C03602=1038.319,72.260,-89.888,169.485,39.498,157.426
C03603=1038.313,72.011,-89.869,169.482,39.498,157.426
C03604=1038.308,71.762,-89.852,169.480,39.497,157.426
C03605=1038.301,71.513,-89.833,169.478,39.498,157.426
C03606=1038.295,71.263,-89.815,169.476,39.497,157.425
C03607=1038.289,71.014,-89.797,169.474,39.497,157.425
C03608=1038.282,70.764,-89.779,169.472,39.497,157.425
C03609=1038.276,70.516,-89.761,169.471,39.496,157.425
C03610=1038.270,70.266,-89.743,169.469,39.496,157.425
C03611=1038.263,70.017,-89.724,169.467,39.496,157.425
C03612=1038.257,69.767,-89.706,169.465,39.495,157.425
C03613=1038.252,69.518,-89.689,169.462,39.495,157.425
C03614=1038.245,69.269,-89.670,169.460,39.495,157.425
C03615=1038.238,69.020,-89.653,169.458,39.495,157.424
C03616=1038.232,68.771,-89.634,169.456,39.494,157.424
C03617=1038.226,68.521,-89.616,169.454,39.494,157.424
C03618=1038.220,68.272,-89.599,169.452,39.494,157.424
C03619=1038.213,68.023,-89.581,169.450,39.494,157.424
C03620=1038.207,67.773,-89.563,169.448,39.493,157.424
C03621=1038.201,67.524,-89.545,169.446,39.493,157.424
C03622=1038.194,67.275,-89.527,169.444,39.493,157.424
C03623=1038.188,67.026,-89.509,169.441,39.493,157.423
C03624=1038.182,66.776,-89.491,169.439,39.493,157.423
C03625=1038.176,66.527,-89.473,169.438,39.492,157.423
C03626=1038.169,66.277,-89.455,169.436,39.492,157.423
C03627=1038.163,66.028,-89.438,169.434,39.492,157.423
C03628=1038.157,65.779,-89.419,169.432,39.491,157.423
C03629=1038.150,65.530,-89.402,169.430,39.492,157.423
C03630=1038.144,65.280,-89.384,169.428,39.491,157.423
C03631=1038.138,65.031,-89.366,169.426,39.491,157.423
C03632=1038.131,64.782,-89.348,169.424,39.491,157.423
C03633=1038.125,64.532,-89.330,169.421,39.490,157.422
C03634=1038.120,64.283,-89.313,169.419,39.490,157.422
C03635=1038.113,64.034,-89.295,169.417,39.490,157.422
C03636=1038.106,63.785,-89.277,169.415,39.489,157.422
C03637=1038.099,63.535,-89.259,169.413,39.490,157.422
C03638=1038.094,63.286,-89.242,169.411,39.489,157.422
C03639=1038.087,63.037,-89.224,169.409,39.489,157.422
C03640=1038.080,62.788,-89.207,169.407,39.489,157.422
C03641=1038.074,62.538,-89.189,169.405,39.489,157.422
C03642=1038.068,62.289,-89.172,169.403,39.488,157.421
C03643=1038.061,62.040,-89.154,169.401,39.489,157.421
C03644=1038.055,61.791,-89.136,169.399,39.488,157.421
C03645=1038.048,61.541,-89.119,169.397,39.488,157.421
C03646=1038.042,61.292,-89.101,169.394,39.488,157.421
C03647=1038.035,61.005,-89.081,169.392,39.488,157.421
C03648=1038.028,60.719,-89.061,169.390,39.487,157.421
C03649=1038.019,60.433,-89.041,169.387,39.488,157.421
C03650=1038.012,60.147,-89.021,169.385,39.487,157.421
C03651=1038.006,59.897,-89.003,169.383,39.487,157.421
C03652=1037.999,59.648,-88.986,169.381,39.487,157.420
C03653=1037.994,59.399,-88.969,169.379,39.487,157.420
C03654=1037.987,59.150,-88.951,169.377,39.487,157.420
C03655=1037.980,58.900,-88.934,169.375,39.487,157.420
C03656=1037.974,58.650,-88.916,169.373,39.486,157.420
C03657=1037.968,58.402,-88.899,169.370,39.486,157.420
C03658=1037.961,58.152,-88.882,169.368,39.486,157.420
C03659=1037.955,57.902,-88.864,169.366,39.486,157.420
C03660=1037.949,57.654,-88.847,169.364,39.486,157.420
C03661=1037.942,57.404,-88.829,169.362,39.486,157.419
C03662=1037.936,57.155,-88.812,169.360,39.485,157.419
C03663=1037.929,56.906,-88.794,169.358,39.485,157.419
C03664=1037.923,56.656,-88.777,169.357,39.485,157.419
C03665=1037.917,56.407,-88.760,169.355,39.485,157.419
C03666=1037.910,56.158,-88.742,169.353,39.485,157.419
C03667=1037.904,55.908,-88.724,169.351,39.485,157.419
C03668=1037.898,55.660,-88.707,169.349,39.484,157.419
C03669=1037.891,55.410,-88.690,169.347,39.484,157.419
C03670=1037.885,55.161,-88.672,169.344,39.484,157.419
C03671=1037.878,54.912,-88.655,169.342,39.483,157.418
C03672=1037.872,54.662,-88.638,169.340,39.484,157.418
C03673=1037.866,54.413,-88.620,169.338,39.483,157.418
C03674=1037.860,54.163,-88.604,169.336,39.483,157.418
C03675=1037.853,53.914,-88.587,169.334,39.483,157.418
C03676=1037.847,53.665,-88.569,169.332,39.483,157.418
C03677=1037.840,53.415,-88.551,169.330,39.482,157.418
C03678=1037.834,53.166,-88.534,169.328,39.483,157.418
C03679=1037.828,52.917,-88.516,169.326,39.482,157.418
C03680=1037.822,52.668,-88.499,169.324,39.482,157.418
C03681=1037.815,52.418,-88.483,169.321,39.482,157.417
C03682=1037.810,52.169,-88.465,169.319,39.481,157.417
C03683=1037.803,51.919,-88.448,169.317,39.481,157.417
C03684=1037.796,51.671,-88.431,169.315,39.481,157.417
C03685=1037.790,51.421,-88.413,169.313,39.481,157.417
C03686=1037.784,51.172,-88.396,169.311,39.481,157.417
C03687=1037.778,50.922,-88.379,169.309,39.481,157.417
C03688=1037.771,50.672,-88.361,169.307,39.480,157.417
C03689=1037.765,50.424,-88.345,169.305,39.480,157.417
C03690=1037.758,50.174,-88.327,169.303,39.480,157.416
C03691=1037.753,49.925,-88.310,169.300,39.479,157.416
C03692=1037.746,49.675,-88.293,169.298,39.480,157.416
C03693=1037.740,49.427,-88.276,169.296,39.479,157.416
C03694=1037.734,49.177,-88.258,169.294,39.479,157.416
C03695=1037.728,48.927,-88.242,169.293,39.479,157.416
C03696=1037.721,48.678,-88.224,169.291,39.478,157.416
C03697=1037.716,48.429,-88.207,169.289,39.478,157.416
C03698=1037.709,48.180,-88.190,169.287,39.478,157.415
C03699=1037.703,47.930,-88.173,169.285,39.478,157.415
C03700=1037.697,47.681,-88.156,169.283,39.478,157.415
C03701=1037.690,47.432,-88.138,169.280,39.477,157.415
C03702=1037.684,47.182,-88.122,169.278,39.477,157.415
C03703=1037.678,46.933,-88.104,169.276,39.477,157.415
C03704=1037.672,46.684,-88.087,169.274,39.477,157.415
C03705=1037.665,46.434,-88.071,169.272,39.476,157.415
C03706=1037.659,46.185,-88.054,169.270,39.476,157.415
C03707=1037.653,45.935,-88.036,169.268,39.476,157.415
C03708=1037.647,45.686,-88.019,169.266,39.476,157.414
C03709=1037.641,45.437,-88.002,169.264,39.476,157.414
C03710=1037.635,45.188,-87.985,169.262,39.475,157.414
C03711=1037.627,44.901,-87.966,169.260,39.475,157.414
C03712=1037.620,44.614,-87.946,169.258,39.475,157.414
C03713=1037.613,44.328,-87.926,169.254,39.474,157.414
C03714=1037.606,44.042,-87.907,169.252,39.474,157.414
C03715=1037.600,43.792,-87.890,169.250,39.474,157.414
C03716=1037.594,43.542,-87.873,169.248,39.474,157.413
C03717=1037.588,43.293,-87.856,169.246,39.473,157.413
C03718=1037.582,43.044,-87.839,169.244,39.473,157.413
C03719=1037.575,42.795,-87.822,169.242,39.473,157.413
C03720=1037.569,42.545,-87.806,169.240,39.473,157.413
C03721=1037.563,42.296,-87.789,169.238,39.472,157.413
C03722=1037.556,42.046,-87.772,169.236,39.473,157.413
C03723=1037.550,41.797,-87.755,169.233,39.472,157.413
C03724=1037.544,41.548,-87.739,169.231,39.472,157.413
C03725=1037.537,41.299,-87.722,169.229,39.472,157.412
C03726=1037.531,41.049,-87.705,169.227,39.472,157.412
C03727=1037.524,40.800,-87.688,169.225,39.471,157.412
C03728=1037.518,40.550,-87.672,169.223,39.472,157.412
C03729=1037.512,40.302,-87.655,169.221,39.471,157.412
C03730=1037.505,40.052,-87.638,169.219,39.471,157.412
C03731=1037.499,39.802,-87.622,169.217,39.471,157.412
C03732=1037.493,39.553,-87.605,169.215,39.471,157.412
C03733=1037.487,39.303,-87.588,169.213,39.470,157.412
C03734=1037.481,39.055,-87.571,169.211,39.471,157.412
C03735=1037.475,38.804,-87.554,169.208,39.470,157.411
C03736=1037.469,38.555,-87.538,169.206,39.470,157.411
C03737=1037.462,38.306,-87.521,169.204,39.470,157.411
C03738=1037.456,38.056,-87.504,169.202,39.470,157.411
C03739=1037.450,37.807,-87.488,169.200,39.469,157.411
C03740=1037.444,37.558,-87.471,169.198,39.470,157.411
C03741=1037.437,37.308,-87.454,169.196,39.469,157.411
C03742=1037.430,37.059,-87.439,169.194,39.469,157.411
C03743=1037.424,36.810,-87.422,169.192,39.469,157.411
C03744=1037.418,36.560,-87.405,169.190,39.469,157.411
C03745=1037.412,36.311,-87.389,169.188,39.469,157.411
C03746=1037.405,36.061,-87.372,169.186,39.469,157.410
C03747=1037.398,35.813,-87.356,169.184,39.469,157.410
C03748=1037.392,35.563,-87.340,169.182,39.469,157.410
C03749=1037.386,35.313,-87.323,169.179,39.468,157.410
C03750=1037.380,35.064,-87.307,169.177,39.469,157.410
C03751=1037.373,34.815,-87.290,169.175,39.468,157.410
C03752=1037.366,34.565,-87.274,169.173,39.468,157.410
C03753=1037.360,34.316,-87.257,169.171,39.468,157.410
C03754=1037.354,34.067,-87.241,169.169,39.468,157.410
C03755=1037.348,33.817,-87.225,169.167,39.468,157.410
C03756=1037.341,33.568,-87.208,169.165,39.468,157.409
C03757=1037.335,33.319,-87.192,169.163,39.468,157.409
C03758=1037.329,33.070,-87.176,169.161,39.467,157.409
C03759=1037.322,32.819,-87.159,169.159,39.467,157.409
C03760=1037.316,32.570,-87.143,169.157,39.468,157.409
C03761=1037.309,32.321,-87.127,169.155,39.467,157.409
C03762=1037.304,32.072,-87.111,169.153,39.467,157.409
C03763=1037.297,31.822,-87.094,169.150,39.467,157.409
C03764=1037.291,31.573,-87.077,169.147,39.467,157.409
C03765=1037.285,31.324,-87.061,169.145,39.466,157.409
C03766=1037.278,31.075,-87.045,169.143,39.467,157.409
C03767=1037.272,30.825,-87.029,169.141,39.467,157.409
C03768=1037.266,30.575,-87.013,169.139,39.466,157.408
C03769=1037.260,30.326,-86.996,169.137,39.466,157.408
C03770=1037.253,30.077,-86.981,169.135,39.466,157.408
C03771=1037.246,29.827,-86.964,169.133,39.466,157.408
C03772=1037.240,29.577,-86.948,169.131,39.466,157.408
C03773=1037.234,29.328,-86.931,169.129,39.466,157.408
C03774=1037.227,29.080,-86.915,169.127,39.466,157.408
C03775=1037.221,28.792,-86.896,169.124,39.465,157.408
C03776=1037.213,28.505,-86.878,169.121,39.465,157.408
C03777=1037.206,28.219,-86.859,169.119,39.465,157.407
C03778=1037.199,27.932,-86.841,169.117,39.465,157.407
C03779=1037.193,27.683,-86.825,169.115,39.465,157.407
C03780=1037.185,27.433,-86.809,169.113,39.465,157.407
C03781=1037.179,27.184,-86.792,169.111,39.464,157.407
C03782=1037.174,26.935,-86.776,169.109,39.465,157.407
C03783=1037.167,26.686,-86.761,169.106,39.465,157.407
C03784=1037.161,26.436,-86.744,169.104,39.464,157.407
C03785=1037.154,26.186,-86.728,169.102,39.464,157.407
C03786=1037.148,25.937,-86.712,169.100,39.465,157.407
C03787=1037.142,25.688,-86.696,169.098,39.464,157.407
C03788=1037.135,25.439,-86.680,169.096,39.464,157.407
C03789=1037.129,25.189,-86.665,169.094,39.464,157.407
C03790=1037.122,24.939,-86.649,169.091,39.464,157.406
C03791=1037.116,24.690,-86.632,169.089,39.464,157.406
C03792=1037.109,24.441,-86.617,169.087,39.464,157.406
C03793=1037.103,24.191,-86.600,169.085,39.464,157.406
C03794=1037.097,23.942,-86.585,169.083,39.464,157.406
C03795=1037.091,23.693,-86.568,169.081,39.464,157.406
C03796=1037.084,23.443,-86.553,169.079,39.464,157.406
C03797=1037.078,23.193,-86.537,169.076,39.464,157.406
C03798=1037.071,22.944,-86.521,169.074,39.464,157.406
C03799=1037.065,22.695,-86.505,169.072,39.463,157.406
C03800=1037.059,22.446,-86.489,169.070,39.464,157.406
C03801=1037.053,22.196,-86.474,169.068,39.463,157.405
C03802=1037.046,21.947,-86.458,169.066,39.463,157.405
C03803=1037.040,21.697,-86.442,169.064,39.463,157.405
C03804=1037.033,21.448,-86.426,169.062,39.463,157.405
C03805=1037.027,21.198,-86.410,169.060,39.463,157.405
C03806=1037.021,20.949,-86.395,169.057,39.463,157.405
C03807=1037.015,20.699,-86.378,169.055,39.463,157.405
C03808=1037.008,20.450,-86.363,169.053,39.463,157.405
C03809=1037.002,20.201,-86.346,169.051,39.462,157.405
C03810=1036.996,19.951,-86.331,169.048,39.463,157.405
C03811=1036.990,19.702,-86.315,169.046,39.463,157.405
C03812=1036.983,19.453,-86.300,169.044,39.462,157.404
C03813=1036.977,19.202,-86.284,169.042,39.462,157.404
C03814=1036.970,18.953,-86.268,169.040,39.463,157.404
C03815=1036.963,18.704,-86.252,169.038,39.463,157.404
C03816=1036.958,18.454,-86.237,169.036,39.462,157.404
C03817=1036.951,18.205,-86.221,169.034,39.462,157.404
C03818=1036.945,17.956,-86.205,169.032,39.463,157.404
C03819=1036.939,17.706,-86.190,169.030,39.462,157.404
C03820=1036.932,17.457,-86.174,169.027,39.462,157.404
C03821=1036.926,17.207,-86.159,169.025,39.463,157.404
C03822=1036.920,16.958,-86.143,169.022,39.462,157.404
C03823=1036.913,16.709,-86.127,169.020,39.462,157.404
C03824=1036.907,16.459,-86.112,169.018,39.462,157.404
C03825=1036.901,16.210,-86.096,169.016,39.462,157.403
C03826=1036.894,15.960,-86.081,169.014,39.462,157.403
C03827=1036.888,15.711,-86.065,169.012,39.462,157.403
C03828=1036.882,15.462,-86.049,169.010,39.462,157.403
C03829=1036.875,15.212,-86.034,169.007,39.462,157.403
C03830=1036.869,14.963,-86.018,169.005,39.462,157.403
C03831=1036.862,14.713,-86.003,169.003,39.462,157.403
C03832=1036.856,14.463,-85.987,169.001,39.462,157.403
C03833=1036.850,14.214,-85.972,168.999,39.462,157.403
C03834=1036.843,13.965,-85.956,168.997,39.462,157.403
C03835=1036.837,13.715,-85.941,168.995,39.461,157.403
C03836=1036.830,13.466,-85.925,168.993,39.462,157.403
C03837=1036.825,13.216,-85.910,168.990,39.462,157.403
C03838=1036.818,12.967,-85.894,168.988,39.462,157.403
C03839=1036.811,12.681,-85.877,168.986,39.462,157.402
C03840=1036.803,12.396,-85.859,168.982,39.462,157.402
C03841=1036.796,12.111,-85.842,168.980,39.462,157.402
C03842=1036.789,11.826,-85.824,168.977,39.462,157.402
C03843=1036.782,11.576,-85.810,168.975,39.462,157.402
C03844=1036.776,11.327,-85.795,168.973,39.462,157.402
C03845=1036.769,11.078,-85.779,168.971,39.462,157.402
C03846=1036.763,10.828,-85.764,168.969,39.462,157.402
C03847=1036.756,10.579,-85.748,168.967,39.462,157.402
C03848=1036.750,10.329,-85.733,168.964,39.463,157.402
C03849=1036.743,10.080,-85.718,168.962,39.463,157.402
C03850=1036.737,9.830,-85.702,168.960,39.462,157.402
C03851=1036.731,9.581,-85.687,168.958,39.462,157.402
C03852=1036.725,9.331,-85.672,168.956,39.462,157.402
C03853=1036.718,9.082,-85.657,168.954,39.463,157.402
C03854=1036.712,8.832,-85.642,168.952,39.463,157.401
C03855=1036.705,8.583,-85.627,168.949,39.462,157.401
C03856=1036.699,8.333,-85.612,168.947,39.463,157.401
C03857=1036.692,8.084,-85.596,168.945,39.463,157.401
C03858=1036.686,7.834,-85.581,168.943,39.463,157.401
C03859=1036.679,7.585,-85.566,168.941,39.463,157.401
C03860=1036.673,7.335,-85.551,168.938,39.462,157.401
C03861=1036.666,7.086,-85.536,168.935,39.463,157.401
C03862=1036.660,6.836,-85.521,168.933,39.463,157.401
C03863=1036.655,6.587,-85.506,168.931,39.463,157.401
C03864=1036.648,6.337,-85.491,168.929,39.463,157.401
C03865=1036.642,6.088,-85.475,168.927,39.463,157.401
C03866=1036.635,5.839,-85.460,168.925,39.463,157.401
C03867=1036.629,5.589,-85.445,168.922,39.463,157.401
C03868=1036.623,5.339,-85.430,168.920,39.463,157.400
C03869=1036.616,5.090,-85.414,168.918,39.463,157.400
C03870=1036.610,4.841,-85.399,168.916,39.463,157.400
C03871=1036.603,4.591,-85.385,168.914,39.463,157.400
C03872=1036.597,4.342,-85.370,168.912,39.463,157.400
C03873=1036.591,4.092,-85.355,168.909,39.463,157.400
C03874=1036.585,3.843,-85.340,168.907,39.463,157.400
C03875=1036.578,3.594,-85.324,168.905,39.463,157.400
C03876=1036.572,3.344,-85.309,168.903,39.463,157.400
C03877=1036.565,3.094,-85.294,168.901,39.463,157.400
C03878=1036.559,2.845,-85.280,168.898,39.463,157.400
C03879=1036.553,2.596,-85.265,168.896,39.463,157.400
C03880=1036.547,2.346,-85.250,168.894,39.463,157.400
C03881=1036.540,2.097,-85.235,168.892,39.463,157.400
C03882=1036.534,1.847,-85.220,168.889,39.463,157.399
C03883=1036.527,1.597,-85.205,168.887,39.463,157.399
C03884=1036.521,1.349,-85.190,168.884,39.463,157.399
C03885=1036.515,1.099,-85.175,168.882,39.463,157.399
C03886=1036.509,0.849,-85.159,168.880,39.463,157.399
C03887=1036.503,0.600,-85.144,168.878,39.463,157.399
C03888=1036.497,0.350,-85.130,168.876,39.463,157.399
C03889=1036.491,0.101,-85.115,168.874,39.463,157.399
C03890=1036.484,-0.149,-85.100,168.871,39.464,157.399
C03891=1036.478,-0.398,-85.085,168.869,39.463,157.399
C03892=1036.472,-0.648,-85.070,168.867,39.463,157.399
C03893=1036.466,-0.897,-85.056,168.865,39.463,157.399
C03894=1036.460,-1.147,-85.041,168.863,39.463,157.399
C03895=1036.453,-1.396,-85.026,168.860,39.463,157.398
C03896=1036.447,-1.646,-85.011,168.858,39.463,157.398
C03897=1036.441,-1.895,-84.996,168.856,39.464,157.398
C03898=1036.435,-2.145,-84.981,168.854,39.463,157.398
C03899=1036.428,-2.394,-84.966,168.852,39.463,157.398
C03900=1036.422,-2.644,-84.951,168.849,39.463,157.398
C03901=1036.416,-2.893,-84.937,168.846,39.464,157.398
C03902=1036.410,-3.142,-84.922,168.844,39.463,157.398
C03903=1036.399,-3.564,-84.897,168.840,39.463,157.398
C03904=1036.388,-3.986,-84.872,168.837,39.464,157.398
C03905=1036.380,-4.308,-84.853,168.834,39.464,157.398
C03906=1036.372,-4.630,-84.835,168.831,39.464,157.398
C03907=1036.364,-4.952,-84.816,168.828,39.464,157.398
C03908=1036.355,-5.275,-84.797,168.825,39.464,157.397
C03909=1036.349,-5.524,-84.783,168.823,39.464,157.397
C03910=1036.342,-5.773,-84.768,168.820,39.464,157.397
C03911=1036.336,-6.023,-84.754,168.818,39.464,157.397
C03912=1036.330,-6.272,-84.739,168.816,39.465,157.397
C03913=1036.323,-6.522,-84.725,168.814,39.465,157.397
C03914=1036.317,-6.771,-84.710,168.811,39.465,157.397
C03915=1036.311,-7.021,-84.696,168.809,39.465,157.397
C03916=1036.304,-7.270,-84.682,168.807,39.465,157.397
C03917=1036.298,-7.520,-84.667,168.805,39.465,157.397
C03918=1036.291,-7.769,-84.652,168.802,39.466,157.397
C03919=1036.285,-8.019,-84.639,168.800,39.466,157.397
C03920=1036.279,-8.268,-84.624,168.798,39.466,157.397
C03921=1036.272,-8.518,-84.609,168.796,39.466,157.397
C03922=1036.266,-8.767,-84.596,168.793,39.466,157.397
C03923=1036.260,-9.017,-84.581,168.791,39.466,157.397
C03924=1036.253,-9.267,-84.566,168.789,39.466,157.397
C03925=1036.247,-9.516,-84.552,168.787,39.466,157.397
C03926=1036.241,-9.766,-84.537,168.784,39.466,157.397
C03927=1036.234,-10.015,-84.522,168.782,39.467,157.396
C03928=1036.228,-10.264,-84.509,168.779,39.467,157.396
C03929=1036.222,-10.514,-84.494,168.777,39.467,157.396
C03930=1036.215,-10.763,-84.480,168.774,39.467,157.396
C03931=1036.209,-11.013,-84.466,168.772,39.467,157.396
C03932=1036.203,-11.263,-84.451,168.770,39.467,157.396
C03933=1036.196,-11.511,-84.437,168.767,39.468,157.396
C03934=1036.190,-11.762,-84.423,168.765,39.467,157.396
C03935=1036.185,-12.011,-84.408,168.763,39.467,157.396
C03936=1036.178,-12.260,-84.395,168.761,39.467,157.396
C03937=1036.171,-12.510,-84.380,168.758,39.468,157.396
C03938=1036.166,-12.760,-84.366,168.756,39.468,157.396
C03939=1036.159,-13.009,-84.352,168.754,39.468,157.396
C03940=1036.153,-13.258,-84.337,168.752,39.468,157.396
C03941=1036.146,-13.508,-84.323,168.749,39.468,157.396
C03942=1036.140,-13.758,-84.308,168.747,39.468,157.396
C03943=1036.134,-14.007,-84.294,168.745,39.469,157.396
C03944=1036.127,-14.257,-84.280,168.742,39.468,157.395
C03945=1036.122,-14.506,-84.266,168.740,39.468,157.395
C03946=1036.115,-14.756,-84.251,168.738,39.469,157.395
C03947=1036.109,-15.005,-84.238,168.736,39.469,157.395
C03948=1036.103,-15.255,-84.223,168.733,39.469,157.395
C03949=1036.096,-15.504,-84.210,168.731,39.469,157.395
C03950=1036.090,-15.754,-84.195,168.729,39.469,157.395
C03951=1036.084,-16.003,-84.182,168.726,39.469,157.395
C03952=1036.078,-16.253,-84.167,168.724,39.470,157.395
C03953=1036.071,-16.503,-84.153,168.722,39.470,157.395
C03954=1036.064,-16.752,-84.140,168.719,39.470,157.395
C03955=1036.058,-17.001,-84.125,168.717,39.470,157.395
C03956=1036.052,-17.251,-84.112,168.715,39.470,157.395
C03957=1036.045,-17.501,-84.098,168.712,39.471,157.395
C03958=1036.039,-17.750,-84.083,168.710,39.471,157.395
C03959=1036.032,-18.000,-84.070,168.708,39.471,157.395
C03960=1036.027,-18.249,-84.056,168.705,39.472,157.395
C03961=1036.020,-18.499,-84.041,168.703,39.472,157.395
C03962=1036.014,-18.748,-84.028,168.701,39.472,157.395
C03963=1036.008,-18.998,-84.014,168.698,39.472,157.395
C03964=1036.001,-19.247,-84.000,168.696,39.472,157.395
C03965=1035.994,-19.529,-83.985,168.693,39.473,157.395
C03966=1035.986,-19.811,-83.969,168.691,39.473,157.395
C03967=1035.980,-20.093,-83.953,168.687,39.473,157.394
C03968=1035.972,-20.375,-83.937,168.684,39.473,157.394
C03969=1035.966,-20.624,-83.924,168.682,39.473,157.394
C03970=1035.960,-20.874,-83.910,168.680,39.474,157.394
C03971=1035.953,-21.123,-83.896,168.677,39.474,157.394
C03972=1035.947,-21.373,-83.882,168.675,39.474,157.394
C03973=1035.941,-21.622,-83.868,168.673,39.474,157.394
C03974=1035.934,-21.872,-83.855,168.670,39.474,157.394
C03975=1035.928,-22.121,-83.840,168.668,39.474,157.394
C03976=1035.922,-22.370,-83.827,168.666,39.475,157.394
C03977=1035.915,-22.620,-83.813,168.663,39.475,157.394
C03978=1035.910,-22.870,-83.799,168.661,39.475,157.394
C03979=1035.903,-23.120,-83.786,168.659,39.475,157.394
C03980=1035.897,-23.369,-83.772,168.656,39.475,157.394
C03981=1035.891,-23.618,-83.758,168.654,39.476,157.394
C03982=1035.884,-23.868,-83.744,168.652,39.476,157.394
C03983=1035.878,-24.117,-83.731,168.649,39.477,157.394
C03984=1035.872,-24.368,-83.717,168.647,39.477,157.394
C03985=1035.866,-24.617,-83.704,168.645,39.477,157.394
C03986=1035.860,-24.866,-83.690,168.642,39.477,157.394
C03987=1035.853,-25.116,-83.675,168.640,39.477,157.394
C03988=1035.847,-25.365,-83.662,168.638,39.477,157.394
C03989=1035.841,-25.614,-83.649,168.635,39.478,157.394
C03990=1035.834,-25.864,-83.635,168.633,39.478,157.394
C03991=1035.829,-26.114,-83.621,168.630,39.478,157.393
C03992=1035.822,-26.364,-83.608,168.628,39.478,157.393
C03993=1035.815,-26.613,-83.594,168.626,39.478,157.393
C03994=1035.810,-26.863,-83.581,168.623,39.479,157.393
C03995=1035.803,-27.113,-83.567,168.621,39.479,157.393
C03996=1035.797,-27.362,-83.554,168.619,39.479,157.393
C03997=1035.791,-27.611,-83.540,168.616,39.479,157.393
C03998=1035.784,-27.861,-83.527,168.614,39.479,157.393
C03999=1035.778,-28.110,-83.513,168.611,39.480,157.393
C04000=1035.772,-28.360,-83.500,168.609,39.480,157.393
C04001=1035.765,-28.610,-83.486,168.607,39.481,157.393
C04002=1035.759,-28.859,-83.473,168.604,39.481,157.393
C04003=1035.752,-29.109,-83.459,168.602,39.481,157.393
C04004=1035.746,-29.358,-83.446,168.599,39.482,157.393
C04005=1035.740,-29.608,-83.432,168.597,39.482,157.393
C04006=1035.733,-29.858,-83.419,168.595,39.482,157.393
C04007=1035.727,-30.107,-83.406,168.592,39.482,157.393
C04008=1035.721,-30.356,-83.392,168.590,39.482,157.393
C04009=1035.715,-30.606,-83.380,168.587,39.483,157.393
C04010=1035.708,-30.856,-83.366,168.585,39.484,157.393
C04011=1035.702,-31.105,-83.353,168.582,39.484,157.393
C04012=1035.696,-31.355,-83.340,168.580,39.484,157.393
C04013=1035.689,-31.605,-83.326,168.578,39.484,157.393
C04014=1035.683,-31.854,-83.313,168.575,39.484,157.393
C04015=1035.676,-32.103,-83.299,168.573,39.485,157.393
C04016=1035.670,-32.353,-83.287,168.570,39.485,157.393
C04017=1035.664,-32.603,-83.273,168.568,39.485,157.393
C04018=1035.658,-32.853,-83.259,168.565,39.486,157.393
C04019=1035.652,-33.102,-83.246,168.563,39.486,157.393
C04020=1035.646,-33.351,-83.233,168.561,39.486,157.393
C04021=1035.639,-33.601,-83.219,168.558,39.487,157.393
C04022=1035.633,-33.851,-83.207,168.556,39.487,157.393
C04023=1035.627,-34.100,-83.193,168.553,39.487,157.393
C04024=1035.621,-34.349,-83.180,168.551,39.487,157.392
C04025=1035.614,-34.599,-83.166,168.548,39.488,157.392
C04026=1035.608,-34.849,-83.154,168.546,39.489,157.393
C04027=1035.602,-35.099,-83.141,168.544,39.489,157.392
C04028=1035.595,-35.348,-83.127,168.541,39.489,157.392
C04029=1035.588,-35.629,-83.113,168.538,39.489,157.392
C04030=1035.581,-35.910,-83.097,168.536,39.489,157.392
C04031=1035.574,-36.191,-83.083,168.533,39.490,157.392
C04032=1035.567,-36.472,-83.069,168.530,39.490,157.392
C04033=1035.561,-36.722,-83.055,168.528,39.491,157.392
C04034=1035.555,-36.971,-83.042,168.525,39.491,157.392
C04035=1035.549,-37.221,-83.030,168.523,39.491,157.392
C04036=1035.542,-37.471,-83.016,168.520,39.491,157.392
C04037=1035.536,-37.720,-83.003,168.518,39.492,157.392
C04038=1035.530,-37.970,-82.990,168.516,39.492,157.392
C04039=1035.524,-38.219,-82.977,168.513,39.492,157.392
C04040=1035.517,-38.469,-82.964,168.511,39.493,157.392
C04041=1035.511,-38.718,-82.951,168.508,39.493,157.392
C04042=1035.505,-38.968,-82.937,168.506,39.494,157.392
C04043=1035.499,-39.218,-82.925,168.503,39.494,157.392
C04044=1035.492,-39.468,-82.912,168.501,39.494,157.392
C04045=1035.486,-39.717,-82.898,168.498,39.495,157.392
C04046=1035.480,-39.966,-82.886,168.496,39.495,157.392
C04047=1035.473,-40.216,-82.873,168.493,39.495,157.392
C04048=1035.467,-40.465,-82.861,168.491,39.496,157.392
C04049=1035.461,-40.715,-82.847,168.488,39.496,157.392
C04050=1035.454,-40.965,-82.835,168.486,39.496,157.392
C04051=1035.448,-41.214,-82.822,168.483,39.497,157.392
C04052=1035.442,-41.464,-82.809,168.481,39.497,157.392
C04053=1035.436,-41.713,-82.796,168.478,39.498,157.392
C04054=1035.429,-41.963,-82.784,168.476,39.499,157.392
C04055=1035.423,-42.212,-82.771,168.473,39.499,157.392
C04056=1035.417,-42.462,-82.758,168.471,39.499,157.392
C04057=1035.411,-42.712,-82.746,168.468,39.500,157.392
C04058=1035.403,-42.962,-82.732,168.466,39.500,157.392
C04059=1035.398,-43.212,-82.720,168.463,39.500,157.392
C04060=1035.391,-43.461,-82.707,168.461,39.501,157.392
C04061=1035.385,-43.711,-82.694,168.458,39.501,157.392
C04062=1035.378,-43.960,-82.681,168.456,39.501,157.392
C04063=1035.373,-44.210,-82.669,168.453,39.502,157.392
C04064=1035.367,-44.459,-82.656,168.451,39.502,157.392
C04065=1035.360,-44.709,-82.643,168.448,39.503,157.392
C04066=1035.354,-44.958,-82.631,168.446,39.503,157.392
C04067=1035.348,-45.208,-82.619,168.443,39.504,157.392
C04068=1035.342,-45.457,-82.605,168.441,39.504,157.392
C04069=1035.336,-45.707,-82.593,168.438,39.505,157.392
C04070=1035.329,-45.957,-82.581,168.436,39.505,157.392
C04071=1035.323,-46.206,-82.567,168.433,39.505,157.392
C04072=1035.317,-46.456,-82.555,168.432,39.506,157.392
C04073=1035.310,-46.706,-82.543,168.429,39.506,157.392
C04074=1035.304,-46.955,-82.530,168.426,39.506,157.392
C04075=1035.298,-47.205,-82.517,168.424,39.507,157.392
C04076=1035.292,-47.455,-82.505,168.422,39.507,157.392
C04077=1035.285,-47.704,-82.492,168.419,39.508,157.392
C04078=1035.279,-47.953,-82.479,168.417,39.508,157.392
C04079=1035.274,-48.203,-82.467,168.414,39.509,157.392
C04080=1035.267,-48.453,-82.455,168.412,39.509,157.392
C04081=1035.261,-48.702,-82.442,168.409,39.510,157.392
C04082=1035.255,-48.952,-82.429,168.406,39.510,157.392
C04083=1035.248,-49.202,-82.417,168.404,39.510,157.392
C04084=1035.242,-49.452,-82.405,168.401,39.511,157.392
C04085=1035.236,-49.701,-82.391,168.399,39.511,157.392
C04086=1035.230,-49.951,-82.379,168.396,39.511,157.391
C04087=1035.223,-50.200,-82.367,168.394,39.512,157.392
C04088=1035.218,-50.450,-82.354,168.391,39.512,157.392
C04089=1035.211,-50.700,-82.342,168.389,39.513,157.391
C04090=1035.206,-50.949,-82.330,168.386,39.513,157.392
C04091=1035.199,-51.198,-82.318,168.384,39.514,157.392
C04092=1035.193,-51.448,-82.305,168.381,39.515,157.392
C04093=1035.185,-51.729,-82.292,168.378,39.515,157.392
C04094=1035.178,-52.011,-82.278,168.375,39.516,157.392
C04095=1035.171,-52.293,-82.264,168.372,39.517,157.392
C04096=1035.163,-52.574,-82.251,168.369,39.517,157.392
C04097=1035.157,-52.824,-82.238,168.367,39.518,157.392
C04098=1035.151,-53.073,-82.226,168.364,39.519,157.392
C04099=1035.144,-53.323,-82.214,168.361,39.519,157.392
C04100=1035.138,-53.573,-82.202,168.359,39.520,157.392
C04101=1035.132,-53.822,-82.190,168.356,39.520,157.392
C04102=1035.125,-54.072,-82.178,168.354,39.521,157.392
C04103=1035.119,-54.322,-82.165,168.352,39.522,157.392
C04104=1035.112,-54.571,-82.153,168.349,39.522,157.392
C04105=1035.106,-54.820,-82.142,168.347,39.523,157.392
C04106=1035.100,-55.070,-82.129,168.344,39.523,157.392
C04107=1035.094,-55.320,-82.117,168.342,39.524,157.392
C04108=1035.087,-55.569,-82.105,168.339,39.525,157.392
C04109=1035.081,-55.819,-82.093,168.336,39.525,157.392
C04110=1035.075,-56.069,-82.081,168.334,39.526,157.392
C04111=1035.068,-56.318,-82.069,168.331,39.526,157.392
C04112=1035.062,-56.568,-82.056,168.328,39.527,157.392
C04113=1035.056,-56.817,-82.045,168.326,39.528,157.392
C04114=1035.050,-57.067,-82.033,168.323,39.528,157.392
C04115=1035.044,-57.317,-82.021,168.321,39.529,157.392
C04116=1035.037,-57.567,-82.009,168.318,39.529,157.392
C04117=1035.030,-57.816,-81.997,168.315,39.530,157.392
C04118=1035.025,-58.066,-81.984,168.313,39.531,157.392
C04119=1035.018,-58.315,-81.973,168.310,39.531,157.392
C04120=1035.012,-58.565,-81.961,168.308,39.532,157.392
C04121=1035.006,-58.815,-81.950,168.305,39.532,157.392
C04122=1035.000,-59.065,-81.937,168.302,39.533,157.392
C04123=1034.993,-59.314,-81.925,168.301,39.534,157.392
C04124=1034.987,-59.563,-81.913,168.298,39.534,157.392
C04125=1034.981,-59.813,-81.901,168.295,39.535,157.392
C04126=1034.975,-60.063,-81.890,168.293,39.535,157.392
C04127=1034.968,-60.313,-81.878,168.290,39.536,157.392
C04128=1034.961,-60.562,-81.866,168.288,39.537,157.392
C04129=1034.956,-60.812,-81.854,168.285,39.537,157.392
C04130=1034.949,-61.061,-81.842,168.282,39.538,157.392
C04131=1034.943,-61.311,-81.830,168.280,39.538,157.392
C04132=1034.937,-61.561,-81.818,168.277,39.539,157.392
C04133=1034.931,-61.810,-81.806,168.274,39.540,157.392
C04134=1034.925,-62.060,-81.795,168.272,39.540,157.392
C04135=1034.918,-62.310,-81.783,168.269,39.541,157.392
C04136=1034.913,-62.559,-81.771,168.266,39.542,157.392
C04137=1034.906,-62.809,-81.759,168.264,39.542,157.392
C04138=1034.900,-63.059,-81.748,168.261,39.543,157.392
C04139=1034.893,-63.308,-81.736,168.259,39.543,157.392
C04140=1034.888,-63.558,-81.723,168.256,39.544,157.392
C04141=1034.882,-63.808,-81.712,168.253,39.545,157.392
C04142=1034.875,-64.057,-81.700,168.251,39.545,157.392
C04143=1034.869,-64.306,-81.689,168.248,39.546,157.392
C04144=1034.863,-64.557,-81.677,168.246,39.546,157.393
C04145=1034.857,-64.806,-81.665,168.244,39.547,157.393
C04146=1034.851,-65.056,-81.654,168.241,39.548,157.393
C04147=1034.844,-65.305,-81.642,168.238,39.548,157.393
C04148=1034.838,-65.555,-81.629,168.236,39.549,157.393
C04149=1034.833,-65.805,-81.619,168.233,39.550,157.393
C04150=1034.826,-66.054,-81.607,168.231,39.550,157.393
C04151=1034.820,-66.304,-81.595,168.228,39.551,157.393
C04152=1034.814,-66.554,-81.583,168.225,39.551,157.393
C04153=1034.808,-66.803,-81.571,168.223,39.552,157.393
C04154=1034.802,-67.053,-81.560,168.220,39.553,157.393
C04155=1034.795,-67.302,-81.548,168.217,39.553,157.393
C04156=1034.790,-67.553,-81.537,168.215,39.554,157.393
C04157=1034.783,-67.835,-81.524,168.212,39.554,157.393
C04158=1034.776,-68.118,-81.511,168.209,39.555,157.393
C04159=1034.769,-68.400,-81.497,168.206,39.556,157.393
C04160=1034.762,-68.683,-81.484,168.203,39.556,157.393
C04161=1034.756,-68.933,-81.473,168.201,39.557,157.393
C04162=1034.749,-69.183,-81.461,168.197,39.558,157.393
C04163=1034.744,-69.432,-81.450,168.196,39.558,157.393
C04164=1034.737,-69.682,-81.438,168.193,39.559,157.393
C04165=1034.732,-69.932,-81.426,168.190,39.560,157.393
C04166=1034.726,-70.182,-81.415,168.188,39.560,157.393
C04167=1034.720,-70.431,-81.404,168.185,39.561,157.393
C04168=1034.713,-70.681,-81.392,168.182,39.562,157.393
C04169=1034.707,-70.930,-81.381,168.180,39.562,157.393
C04170=1034.702,-71.180,-81.369,168.177,39.563,157.393
C04171=1034.696,-71.429,-81.357,168.174,39.564,157.393
C04172=1034.689,-71.679,-81.346,168.172,39.564,157.393
C04173=1034.683,-71.929,-81.335,168.169,39.565,157.393
C04174=1034.677,-72.178,-81.323,168.166,39.565,157.393
C04175=1034.672,-72.428,-81.312,168.164,39.566,157.393
C04176=1034.666,-72.678,-81.300,168.161,39.567,157.393
C04177=1034.659,-72.927,-81.289,168.158,39.567,157.393
C04178=1034.653,-73.177,-81.278,168.156,39.568,157.393
C04179=1034.647,-73.426,-81.266,168.153,39.568,157.393
C04180=1034.641,-73.677,-81.254,168.151,39.569,157.393
C04181=1034.636,-73.926,-81.243,168.149,39.570,157.393
C04182=1034.629,-74.176,-81.232,168.146,39.570,157.393
C04183=1034.623,-74.425,-81.220,168.143,39.571,157.393
C04184=1034.617,-74.675,-81.209,168.141,39.572,157.393
C04185=1034.611,-74.925,-81.198,168.138,39.572,157.393
C04186=1034.605,-75.175,-81.187,168.135,39.573,157.393
C04187=1034.598,-75.424,-81.176,168.132,39.574,157.393
C04188=1034.592,-75.674,-81.165,168.130,39.575,157.394
C04189=1034.586,-75.923,-81.154,168.127,39.576,157.394
C04190=1034.580,-76.174,-81.143,168.124,39.577,157.394
C04191=1034.574,-76.423,-81.132,168.122,39.577,157.394
C04192=1034.568,-76.673,-81.121,168.119,39.578,157.394
C04193=1034.562,-76.922,-81.109,168.116,39.579,157.394
C04194=1034.556,-77.172,-81.098,168.114,39.580,157.394
C04195=1034.550,-77.422,-81.087,168.112,39.581,157.394
C04196=1034.544,-77.671,-81.076,168.109,39.581,157.394
C04197=1034.537,-77.921,-81.065,168.106,39.582,157.394
C04198=1034.531,-78.171,-81.055,168.103,39.583,157.394
C04199=1034.525,-78.420,-81.044,168.101,39.583,157.394
C04200=1034.519,-78.670,-81.032,168.098,39.584,157.394
C04201=1034.513,-78.919,-81.021,168.095,39.585,157.394
C04202=1034.506,-79.169,-81.010,168.093,39.586,157.394
C04203=1034.501,-79.419,-80.999,168.090,39.587,157.394
C04204=1034.495,-79.668,-80.988,168.087,39.588,157.394
C04205=1034.489,-79.919,-80.977,168.084,39.588,157.394
C04206=1034.482,-80.168,-80.966,168.082,39.589,157.394
C04207=1034.476,-80.418,-80.955,168.080,39.590,157.394
C04208=1034.470,-80.667,-80.944,168.077,39.591,157.394
C04209=1034.464,-80.917,-80.934,168.074,39.592,157.394
C04210=1034.457,-81.167,-80.923,168.071,39.593,157.395
C04211=1034.452,-81.416,-80.912,168.069,39.594,157.395
///RCONF 1,0,0,0,1,0,0,0,0,0,0,0,0,0,0,0,0,0,0,0,0,0,0,0
C04212=1034.444,-81.666,-80.901,168.066,39.595,157.395
C04213=1034.439,-81.916,-80.890,168.063,39.596,157.395
C04214=1034.433,-82.165,-80.879,168.060,39.597,157.395
C04215=1034.426,-82.416,-80.869,168.057,39.598,157.395
C04216=1034.420,-82.665,-80.859,168.056,39.598,157.395
C04217=1034.414,-82.914,-80.848,168.053,39.599,157.395
C04218=1034.408,-83.164,-80.837,168.050,39.600,157.395
C04219=1034.402,-83.414,-80.826,168.047,39.601,157.395
C04220=1034.395,-83.663,-80.816,168.045,39.602,157.395
C04221=1034.388,-83.948,-80.804,168.041,39.603,157.395
C04222=1034.381,-84.233,-80.792,168.038,39.604,157.395
C04223=1034.374,-84.518,-80.779,168.035,39.605,157.395
C04224=1034.367,-84.803,-80.767,168.032,39.606,157.396
C04225=1034.361,-85.053,-80.756,168.030,39.607,157.396
C04226=1034.355,-85.303,-80.745,168.027,39.608,157.396
C04227=1034.349,-85.552,-80.735,168.024,39.609,157.396
C04228=1034.343,-85.801,-80.724,168.022,39.610,157.396
C04229=1034.336,-86.052,-80.714,168.019,39.611,157.396
C04230=1034.331,-86.301,-80.703,168.016,39.612,157.396
C04231=1034.325,-86.551,-80.692,168.013,39.613,157.396
C04232=1034.318,-86.801,-80.682,168.010,39.613,157.396
C04233=1034.312,-87.051,-80.672,168.008,39.614,157.396
C04234=1034.306,-87.300,-80.661,168.005,39.615,157.396
C04235=1034.300,-87.550,-80.650,168.003,39.616,157.396
C04236=1034.294,-87.800,-80.639,168.000,39.617,157.396
C04237=1034.288,-88.050,-80.630,167.997,39.618,157.396
C04238=1034.282,-88.299,-80.619,167.995,39.619,157.397
C04239=1034.275,-88.548,-80.608,167.992,39.620,157.397
C04240=1034.270,-88.798,-80.598,167.989,39.621,157.397
C04241=1034.264,-89.049,-80.587,167.986,39.622,157.397
C04242=1034.257,-89.298,-80.577,167.983,39.623,157.397
C04243=1034.251,-89.547,-80.566,167.981,39.624,157.397
C04244=1034.245,-89.797,-80.556,167.979,39.625,157.397
C04245=1034.239,-90.047,-80.545,167.976,39.626,157.397
C04246=1034.232,-90.296,-80.535,167.973,39.627,157.397
C04247=1034.227,-90.547,-80.525,167.970,39.628,157.397
C04248=1034.221,-90.796,-80.514,167.968,39.628,157.397
C04249=1034.215,-91.046,-80.504,167.965,39.629,157.397
C04250=1034.209,-91.295,-80.493,167.962,39.630,157.397
C04251=1034.203,-91.544,-80.483,167.959,39.632,157.397
C04252=1034.197,-91.795,-80.473,167.956,39.633,157.397
C04253=1034.190,-92.044,-80.462,167.955,39.633,157.398
C04254=1034.185,-92.295,-80.452,167.952,39.634,157.398
C04255=1034.179,-92.544,-80.441,167.949,39.635,157.398
C04256=1034.173,-92.793,-80.431,167.946,39.636,157.398
C04257=1034.167,-93.043,-80.421,167.943,39.637,157.398
C04258=1034.161,-93.293,-80.410,167.940,39.638,157.398
C04259=1034.155,-93.543,-80.400,167.938,39.639,157.398
C04260=1034.149,-93.792,-80.390,167.935,39.640,157.398
C04261=1034.143,-94.043,-80.380,167.932,39.641,157.398
C04262=1034.136,-94.292,-80.369,167.930,39.642,157.398
C04263=1034.131,-94.542,-80.359,167.927,39.643,157.398
C04264=1034.125,-94.791,-80.348,167.925,39.644,157.398
C04265=1034.119,-95.041,-80.339,167.922,39.645,157.398
C04266=1034.113,-95.291,-80.328,167.919,39.646,157.398
C04267=1034.107,-95.540,-80.318,167.916,39.647,157.398
C04268=1034.101,-95.790,-80.307,167.913,39.648,157.398
C04269=1034.095,-96.040,-80.298,167.911,39.648,157.399
C04270=1034.089,-96.289,-80.287,167.908,39.650,157.399
C04271=1034.083,-96.539,-80.277,167.906,39.651,157.399
C04272=1034.078,-96.789,-80.267,167.903,39.652,157.399
C04273=1034.071,-97.038,-80.257,167.900,39.653,157.399
C04274=1034.066,-97.288,-80.247,167.897,39.654,157.399
C04275=1034.059,-97.538,-80.236,167.895,39.655,157.399
C04276=1034.054,-97.788,-80.226,167.892,39.655,157.399
C04277=1034.048,-98.038,-80.217,167.889,39.657,157.399
C04278=1034.041,-98.287,-80.206,167.886,39.658,157.399
C04279=1034.035,-98.538,-80.196,167.883,39.659,157.399
C04280=1034.029,-98.787,-80.186,167.881,39.660,157.400
C04281=1034.023,-99.037,-80.176,167.878,39.661,157.400
C04282=1034.016,-99.286,-80.166,167.876,39.662,157.400
C04283=1034.011,-99.536,-80.156,167.873,39.664,157.400
C04284=1034.005,-99.786,-80.147,167.870,39.665,157.400
C04285=1033.998,-100.073,-80.136,167.866,39.666,157.400
C04286=1033.991,-100.360,-80.123,167.864,39.667,157.400
C04287=1033.984,-100.647,-80.112,167.861,39.668,157.400
C04288=1033.977,-100.934,-80.101,167.858,39.670,157.400
C04289=1033.971,-101.184,-80.092,167.855,39.671,157.400
C04290=1033.966,-101.434,-80.081,167.852,39.672,157.401
C04291=1033.959,-101.683,-80.072,167.849,39.673,157.401
C04292=1033.953,-101.933,-80.062,167.846,39.674,157.401
C04293=1033.947,-102.182,-80.052,167.844,39.676,157.401
C04294=1033.941,-102.433,-80.042,167.841,39.677,157.401
C04295=1033.935,-102.682,-80.032,167.838,39.677,157.401
C04296=1033.929,-102.932,-80.023,167.836,39.679,157.401
C04297=1033.923,-103.181,-80.012,167.833,39.680,157.401
C04298=1033.917,-103.431,-80.002,167.830,39.681,157.401
C04299=1033.911,-103.681,-79.993,167.827,39.682,157.401
C04300=1033.905,-103.931,-79.983,167.825,39.683,157.401
C04301=1033.899,-104.181,-79.974,167.822,39.684,157.401
C04302=1033.893,-104.431,-79.963,167.819,39.686,157.402
C04303=1033.888,-104.680,-79.954,167.816,39.687,157.402
C04304=1033.881,-104.930,-79.945,167.813,39.688,157.402
C04305=1033.875,-105.180,-79.935,167.811,39.689,157.402
C04306=1033.869,-105.429,-79.926,167.808,39.690,157.402
C04307=1033.863,-105.679,-79.915,167.806,39.692,157.402
C04308=1033.857,-105.929,-79.905,167.803,39.693,157.402
C04309=1033.851,-106.179,-79.896,167.800,39.693,157.402
C04310=1033.845,-106.428,-79.886,167.797,39.695,157.402
C04311=1033.839,-106.677,-79.877,167.794,39.696,157.402
C04312=1033.833,-106.927,-79.867,167.791,39.698,157.403
C04313=1033.828,-107.177,-79.857,167.788,39.698,157.403
C04314=1033.822,-107.427,-79.847,167.787,39.699,157.403
C04315=1033.815,-107.677,-79.838,167.784,39.701,157.403
C04316=1033.809,-107.927,-79.828,167.781,39.702,157.403
C04317=1033.803,-108.177,-79.819,167.778,39.703,157.403
C04318=1033.798,-108.426,-79.810,167.775,39.704,157.403
C04319=1033.792,-108.676,-79.801,167.772,39.706,157.403
C04320=1033.785,-108.926,-79.791,167.770,39.707,157.403
C04321=1033.779,-109.176,-79.782,167.767,39.708,157.404
C04322=1033.773,-109.425,-79.772,167.764,39.709,157.404
C04323=1033.767,-109.675,-79.762,167.761,39.711,157.404
C04324=1033.761,-109.924,-79.753,167.758,39.712,157.404
C04325=1033.755,-110.174,-79.744,167.755,39.713,157.404
C04326=1033.749,-110.424,-79.734,167.753,39.714,157.404
C04327=1033.743,-110.674,-79.725,167.751,39.716,157.404
C04328=1033.737,-110.924,-79.716,167.748,39.717,157.404
C04329=1033.731,-111.173,-79.706,167.745,39.718,157.404
C04330=1033.725,-111.423,-79.697,167.742,39.719,157.405
C04331=1033.719,-111.673,-79.687,167.739,39.721,157.405
C04332=1033.713,-111.923,-79.678,167.736,39.722,157.405
C04333=1033.708,-112.172,-79.669,167.734,39.723,157.405
C04334=1033.701,-112.422,-79.660,167.731,39.725,157.405
C04335=1033.695,-112.672,-79.650,167.728,39.726,157.405
C04336=1033.689,-112.922,-79.641,167.725,39.727,157.405
C04337=1033.683,-113.171,-79.631,167.722,39.728,157.405
C04338=1033.678,-113.421,-79.623,167.720,39.730,157.406
C04339=1033.671,-113.671,-79.613,167.718,39.731,157.406
C04340=1033.666,-113.920,-79.604,167.715,39.732,157.406
C04341=1033.660,-114.171,-79.595,167.712,39.733,157.406
C04342=1033.654,-114.420,-79.585,167.709,39.735,157.406
C04343=1033.648,-114.670,-79.576,167.706,39.736,157.406
C04344=1033.642,-114.919,-79.567,167.704,39.737,157.406
C04345=1033.636,-115.170,-79.558,167.701,39.739,157.406
C04346=1033.630,-115.419,-79.548,167.698,39.740,157.406
C04347=1033.624,-115.669,-79.539,167.695,39.741,157.407
C04348=1033.619,-115.919,-79.530,167.692,39.743,157.407
C04349=1033.611,-116.205,-79.520,167.689,39.744,157.407
C04350=1033.604,-116.492,-79.509,167.686,39.746,157.407
C04351=1033.598,-116.778,-79.498,167.683,39.747,157.407
C04352=1033.591,-117.065,-79.489,167.680,39.749,157.407
C04353=1033.585,-117.315,-79.479,167.677,39.750,157.407
C04354=1033.579,-117.564,-79.470,167.674,39.751,157.408
C04355=1033.574,-117.814,-79.461,167.672,39.753,157.408
C04356=1033.567,-118.064,-79.452,167.669,39.755,157.408
C04357=1033.562,-118.314,-79.443,167.666,39.755,157.408
C04358=1033.555,-118.563,-79.434,167.663,39.757,157.408
C04359=1033.549,-118.813,-79.425,167.660,39.759,157.408
C04360=1033.543,-119.063,-79.416,167.657,39.760,157.408
C04361=1033.538,-119.312,-79.407,167.655,39.761,157.408
C04362=1033.532,-119.563,-79.398,167.652,39.763,157.409
C04363=1033.525,-119.812,-79.389,167.649,39.764,157.409
C04364=1033.520,-120.062,-79.380,167.646,39.765,157.409
C04365=1033.513,-120.312,-79.371,167.643,39.767,157.409
C04366=1033.508,-120.561,-79.362,167.641,39.768,157.409
C04367=1033.502,-120.812,-79.353,167.638,39.769,157.409
C04368=1033.497,-121.061,-79.344,167.635,39.771,157.409
C04369=1033.490,-121.311,-79.336,167.632,39.773,157.410
C04370=1033.484,-121.561,-79.326,167.629,39.774,157.410
C04371=1033.479,-121.811,-79.318,167.627,39.775,157.410
C04372=1033.473,-122.060,-79.308,167.624,39.777,157.410
C04373=1033.467,-122.310,-79.300,167.621,39.778,157.410
C04374=1033.460,-122.560,-79.291,167.618,39.779,157.410
C04375=1033.455,-122.809,-79.282,167.615,39.781,157.410
C04376=1033.449,-123.060,-79.274,167.613,39.782,157.410
C04377=1033.443,-123.309,-79.265,167.610,39.784,157.411
C04378=1033.437,-123.559,-79.256,167.608,39.785,157.411
C04379=1033.432,-123.809,-79.248,167.605,39.786,157.411
C04380=1033.426,-124.058,-79.238,167.602,39.788,157.411
C04381=1033.420,-124.308,-79.230,167.600,39.790,157.411
C04382=1033.414,-124.558,-79.221,167.597,39.791,157.411
C04383=1033.408,-124.807,-79.212,167.594,39.792,157.411
C04384=1033.402,-125.057,-79.204,167.591,39.794,157.412
C04385=1033.396,-125.307,-79.195,167.588,39.795,157.412
C04386=1033.390,-125.557,-79.186,167.586,39.797,157.412
C04387=1033.384,-125.806,-79.178,167.583,39.799,157.412
C04388=1033.378,-126.057,-79.169,167.580,39.800,157.412
C04389=1033.372,-126.306,-79.161,167.577,39.801,157.412
C04390=1033.366,-126.556,-79.152,167.574,39.803,157.412
C04391=1033.361,-126.806,-79.143,167.572,39.804,157.413
C04392=1033.354,-127.056,-79.135,167.569,39.806,157.413
C04393=1033.349,-127.306,-79.126,167.566,39.808,157.413
C04394=1033.342,-127.555,-79.117,167.563,39.809,157.413
C04395=1033.337,-127.805,-79.109,167.560,39.811,157.413
C04396=1033.332,-128.054,-79.100,167.558,39.812,157.413
C04397=1033.327,-128.304,-79.091,167.555,39.813,157.413
C04398=1033.323,-128.554,-79.080,167.553,39.813,157.413
C04399=1033.319,-128.804,-79.069,167.549,39.812,157.413
C04400=1033.316,-129.053,-79.059,167.547,39.812,157.413
C04401=1033.315,-129.304,-79.046,167.545,39.811,157.413
C04402=1033.313,-129.553,-79.034,167.543,39.809,157.412
C04403=1033.312,-129.803,-79.021,167.541,39.807,157.412
C04404=1033.312,-130.053,-79.007,167.539,39.805,157.412
C04405=1033.313,-130.303,-78.993,167.537,39.802,157.411
C04406=1033.315,-130.553,-78.978,167.535,39.798,157.410
C04407=1033.316,-130.802,-78.963,167.534,39.794,157.410
C04408=1033.320,-131.052,-78.947,167.533,39.790,157.409
C04409=1033.322,-131.303,-78.930,167.531,39.786,157.408
C04410=1033.327,-131.553,-78.914,167.530,39.780,157.407
C04411=1033.331,-131.802,-78.895,167.529,39.775,157.406
C04412=1033.337,-132.053,-78.878,167.528,39.768,157.405
C04413=1033.008,-132.077,-79.166,167.479,39.995,157.441
C04414=1033.002,-131.827,-79.184,167.480,40.001,157.442
C04415=1032.998,-131.578,-79.203,167.481,40.006,157.443
C04416=1032.994,-131.327,-79.220,167.482,40.011,157.444
C04417=1032.991,-131.077,-79.236,167.483,40.016,157.445
C04418=1032.988,-130.828,-79.252,167.485,40.021,157.446
C04419=1032.986,-130.578,-79.267,167.487,40.025,157.446
C04420=1032.984,-130.327,-79.282,167.489,40.028,157.447
C04421=1032.984,-130.077,-79.296,167.490,40.031,157.447
C04422=1032.984,-129.827,-79.310,167.493,40.033,157.448
C04423=1032.985,-129.577,-79.323,167.494,40.035,157.448
C04424=1032.986,-129.328,-79.336,167.497,40.037,157.449
C04425=1032.988,-129.078,-79.347,167.499,40.038,157.449
C04426=1032.991,-128.828,-79.358,167.501,40.039,157.449
C04427=1032.994,-128.579,-79.369,167.503,40.039,157.449
C04428=1032.998,-128.329,-79.379,167.506,40.038,157.449
C04429=1033.003,-128.079,-79.389,167.508,40.038,157.449
C04430=1033.008,-127.830,-79.398,167.511,40.037,157.449
C04431=1033.014,-127.579,-79.406,167.514,40.035,157.449
C04432=1033.020,-127.331,-79.415,167.517,40.033,157.449
C04433=1033.025,-127.081,-79.424,167.519,40.032,157.449
C04434=1033.031,-126.830,-79.432,167.522,40.030,157.449
C04435=1033.037,-126.582,-79.441,167.525,40.029,157.449
C04436=1033.043,-126.331,-79.450,167.528,40.028,157.448
C04437=1033.049,-126.082,-79.458,167.531,40.026,157.448
C04438=1033.055,-125.831,-79.467,167.533,40.024,157.448
C04439=1033.061,-125.582,-79.476,167.537,40.023,157.448
C04440=1033.067,-125.332,-79.484,167.540,40.021,157.448
C04441=1033.073,-125.082,-79.493,167.543,40.019,157.448
C04442=1033.078,-124.832,-79.501,167.545,40.018,157.447
C04443=1033.085,-124.583,-79.510,167.548,40.016,157.447
C04444=1033.091,-124.333,-79.519,167.551,40.014,157.447
C04445=1033.096,-124.083,-79.527,167.554,40.014,157.447
C04446=1033.103,-123.834,-79.536,167.557,40.012,157.447
C04447=1033.108,-123.584,-79.545,167.559,40.010,157.447
C04448=1033.114,-123.334,-79.554,167.562,40.009,157.447
C04449=1033.120,-123.084,-79.563,167.565,40.008,157.447
C04450=1033.126,-122.834,-79.571,167.568,40.006,157.446
C04451=1033.131,-122.585,-79.580,167.571,40.005,157.446
C04452=1033.138,-122.335,-79.589,167.573,40.003,157.446
C04453=1033.143,-122.085,-79.598,167.576,40.001,157.446
C04454=1033.150,-121.836,-79.607,167.578,40.000,157.446
C04455=1033.155,-121.586,-79.615,167.581,39.999,157.446
C04456=1033.161,-121.336,-79.625,167.584,39.997,157.446
C04457=1033.167,-121.086,-79.634,167.586,39.996,157.445
C04458=1033.173,-120.836,-79.641,167.589,39.995,157.445
C04459=1033.179,-120.586,-79.651,167.592,39.993,157.445
C04460=1033.185,-120.337,-79.659,167.595,39.991,157.445
C04461=1033.191,-120.087,-79.669,167.598,39.990,157.445
C04462=1033.196,-119.837,-79.678,167.600,39.989,157.445
C04463=1033.202,-119.587,-79.687,167.603,39.987,157.445
C04464=1033.209,-119.337,-79.695,167.606,39.986,157.444
C04465=1033.214,-119.088,-79.705,167.609,39.984,157.444
C04466=1033.220,-118.838,-79.713,167.612,39.983,157.444
C04467=1033.226,-118.588,-79.723,167.614,39.981,157.444
C04468=1033.232,-118.338,-79.731,167.617,39.980,157.444
C04469=1033.238,-118.089,-79.740,167.620,39.978,157.444
C04470=1033.244,-117.839,-79.749,167.623,39.977,157.444
C04471=1033.250,-117.589,-79.758,167.626,39.976,157.444
C04472=1033.256,-117.340,-79.768,167.628,39.974,157.443
C04473=1033.261,-117.090,-79.777,167.631,39.973,157.443
C04474=1033.269,-116.803,-79.787,167.635,39.971,157.443
C04475=1033.276,-116.517,-79.798,167.638,39.970,157.443
C04476=1033.282,-116.230,-79.809,167.641,39.968,157.443
C04477=1033.289,-115.943,-79.818,167.644,39.967,157.443
C04478=1033.295,-115.694,-79.827,167.647,39.965,157.443
C04479=1033.301,-115.444,-79.837,167.650,39.963,157.442
C04480=1033.307,-115.194,-79.846,167.653,39.962,157.442
C04481=1033.313,-114.945,-79.855,167.656,39.961,157.442
C04482=1033.319,-114.695,-79.865,167.658,39.959,157.442
C04483=1033.325,-114.445,-79.873,167.661,39.958,157.442
C04484=1033.330,-114.196,-79.883,167.664,39.957,157.442
C04485=1033.336,-113.946,-79.892,167.667,39.956,157.442
C04486=1033.342,-113.695,-79.901,167.669,39.954,157.442
C04487=1033.348,-113.446,-79.911,167.671,39.953,157.441
C04488=1033.354,-113.197,-79.920,167.674,39.952,157.441
C04489=1033.360,-112.947,-79.929,167.677,39.950,157.441
C04490=1033.366,-112.696,-79.938,167.680,39.949,157.441
C04491=1033.372,-112.447,-79.947,167.683,39.947,157.441
C04492=1033.378,-112.197,-79.957,167.686,39.946,157.441
C04493=1033.384,-111.948,-79.966,167.688,39.945,157.441
C04494=1033.390,-111.698,-79.976,167.691,39.943,157.441
C04495=1033.395,-111.448,-79.985,167.694,39.942,157.441
C04496=1033.402,-111.198,-79.994,167.697,39.941,157.440
C04497=1033.408,-110.949,-80.004,167.700,39.940,157.440
C04498=1033.414,-110.699,-80.013,167.703,39.938,157.440
C04499=1033.420,-110.449,-80.023,167.705,39.937,157.440
C04500=1033.426,-110.200,-80.032,167.708,39.936,157.440
C04501=1033.431,-109.949,-80.041,167.711,39.934,157.440
C04502=1033.438,-109.700,-80.050,167.714,39.933,157.440
C04503=1033.444,-109.450,-80.060,167.717,39.932,157.440
C04504=1033.450,-109.200,-80.070,167.720,39.931,157.440
C04505=1033.456,-108.951,-80.079,167.721,39.929,157.439
C04506=1033.462,-108.701,-80.088,167.724,39.928,157.439
C04507=1033.468,-108.451,-80.098,167.727,39.927,157.439
C04508=1033.474,-108.202,-80.107,167.730,39.926,157.439
C04509=1033.480,-107.952,-80.117,167.733,39.924,157.439
C04510=1033.486,-107.702,-80.127,167.735,39.922,157.439
C04511=1033.492,-107.453,-80.136,167.738,39.921,157.439
C04512=1033.498,-107.202,-80.145,167.741,39.920,157.439
C04513=1033.503,-106.952,-80.155,167.744,39.919,157.439
C04514=1033.509,-106.703,-80.164,167.747,39.918,157.438
C04515=1033.516,-106.453,-80.174,167.750,39.916,157.438
C04516=1033.522,-106.203,-80.184,167.753,39.915,157.438
C04517=1033.528,-105.954,-80.193,167.755,39.914,157.438
C04518=1033.534,-105.705,-80.203,167.758,39.913,157.438
C04519=1033.539,-105.455,-80.213,167.760,39.911,157.438
C04520=1033.545,-105.205,-80.223,167.763,39.910,157.438
C04521=1033.552,-104.955,-80.232,167.766,39.909,157.438
C04522=1033.558,-104.705,-80.242,167.769,39.908,157.438
C04523=1033.564,-104.455,-80.251,167.772,39.907,157.438
C04524=1033.569,-104.205,-80.262,167.774,39.905,157.437
C04525=1033.576,-103.955,-80.271,167.777,39.904,157.437
C04526=1033.581,-103.706,-80.280,167.780,39.903,157.437
C04527=1033.587,-103.457,-80.290,167.783,39.902,157.437
C04528=1033.593,-103.206,-80.300,167.786,39.901,157.437
C04529=1033.599,-102.957,-80.310,167.788,39.899,157.437
C04530=1033.605,-102.707,-80.320,167.790,39.899,157.437
C04531=1033.612,-102.458,-80.330,167.793,39.897,157.437
C04532=1033.617,-102.208,-80.340,167.796,39.896,157.437
C04533=1033.623,-101.958,-80.349,167.799,39.895,157.437
C04534=1033.629,-101.708,-80.359,167.802,39.893,157.436
C04535=1033.636,-101.459,-80.369,167.805,39.893,157.436
C04536=1033.641,-101.209,-80.379,167.808,39.892,157.436
C04537=1033.647,-100.959,-80.389,167.810,39.890,157.436
C04538=1033.654,-100.672,-80.400,167.813,39.889,157.436
C04539=1033.661,-100.385,-80.411,167.816,39.887,157.436
C04540=1033.668,-100.097,-80.423,167.820,39.886,157.436
C04541=1033.675,-99.811,-80.434,167.823,39.885,157.436
C04542=1033.681,-99.562,-80.444,167.825,39.883,157.436
C04543=1033.687,-99.312,-80.453,167.828,39.882,157.436
C04544=1033.693,-99.062,-80.464,167.831,39.881,157.435
C04545=1033.699,-98.812,-80.474,167.834,39.880,157.435
C04546=1033.705,-98.563,-80.483,167.836,39.879,157.435
C04547=1033.711,-98.312,-80.494,167.839,39.878,157.435
C04548=1033.718,-98.062,-80.504,167.842,39.876,157.435
C04549=1033.724,-97.813,-80.514,167.844,39.876,157.435
C04550=1033.730,-97.563,-80.523,167.847,39.875,157.435
C04551=1033.736,-97.313,-80.534,167.850,39.873,157.435
C04552=1033.741,-97.063,-80.544,167.853,39.872,157.435
C04553=1033.748,-96.814,-80.554,167.856,39.871,157.435
C04554=1033.753,-96.564,-80.565,167.858,39.870,157.435
C04555=1033.760,-96.314,-80.574,167.861,39.869,157.435
C04556=1033.765,-96.064,-80.585,167.864,39.868,157.434
C04557=1033.771,-95.815,-80.595,167.866,39.867,157.434
C04558=1033.777,-95.565,-80.605,167.869,39.866,157.434
C04559=1033.783,-95.316,-80.615,167.872,39.865,157.434
C04560=1033.789,-95.066,-80.626,167.874,39.864,157.434
C04561=1033.795,-94.816,-80.636,167.877,39.863,157.434
C04562=1033.801,-94.566,-80.646,167.880,39.862,157.434
C04563=1033.807,-94.317,-80.656,167.883,39.861,157.434
C04564=1033.813,-94.067,-80.666,167.886,39.860,157.434
C04565=1033.819,-93.818,-80.677,167.888,39.859,157.434
C04566=1033.825,-93.568,-80.687,167.890,39.858,157.434
C04567=1033.831,-93.318,-80.698,167.893,39.857,157.434
C04568=1033.837,-93.068,-80.708,167.896,39.856,157.434
C04569=1033.843,-92.818,-80.719,167.899,39.855,157.433
C04570=1033.849,-92.569,-80.728,167.902,39.854,157.433
C04571=1033.855,-92.319,-80.739,167.905,39.853,157.433
C04572=1033.861,-92.070,-80.749,167.907,39.852,157.433
C04573=1033.867,-91.820,-80.759,167.910,39.851,157.433
C04574=1033.873,-91.571,-80.770,167.912,39.850,157.433
C04575=1033.879,-91.320,-80.780,167.915,39.849,157.433
C04576=1033.885,-91.070,-80.791,167.918,39.847,157.433
C04577=1033.891,-90.821,-80.801,167.921,39.847,157.433
C04578=1033.897,-90.571,-80.812,167.923,39.846,157.433
C04579=1033.903,-90.322,-80.822,167.926,39.845,157.433
C04580=1033.909,-90.072,-80.832,167.929,39.844,157.433
C04581=1033.916,-89.822,-80.843,167.932,39.843,157.433
C04582=1033.922,-89.572,-80.854,167.935,39.842,157.433
C04583=1033.927,-89.322,-80.864,167.937,39.841,157.433
C04584=1033.933,-89.073,-80.874,167.939,39.840,157.432
C04585=1033.939,-88.824,-80.885,167.942,39.839,157.432
C04586=1033.946,-88.573,-80.895,167.945,39.838,157.432
C04587=1033.952,-88.324,-80.906,167.948,39.837,157.432
C04588=1033.957,-88.074,-80.917,167.951,39.836,157.432
C04589=1033.964,-87.825,-80.927,167.954,39.835,157.432
C04590=1033.969,-87.575,-80.937,167.956,39.834,157.432
C04591=1033.976,-87.325,-80.948,167.958,39.833,157.432
C04592=1033.982,-87.075,-80.959,167.961,39.832,157.432
C04593=1033.988,-86.825,-80.969,167.964,39.831,157.432
C04594=1033.994,-86.576,-80.979,167.967,39.830,157.432
C04595=1034.000,-86.326,-80.990,167.970,39.829,157.432
C04596=1034.007,-86.077,-81.000,167.972,39.828,157.432
C04597=1034.013,-85.827,-81.011,167.975,39.827,157.432
C04598=1034.018,-85.577,-81.022,167.978,39.826,157.432
C04599=1034.025,-85.327,-81.032,167.981,39.825,157.431
C04600=1034.031,-85.078,-81.043,167.983,39.824,157.431
C04601=1034.037,-84.829,-81.053,167.985,39.823,157.431
C04602=1034.045,-84.543,-81.066,167.989,39.822,157.431
C04603=1034.051,-84.259,-81.078,167.992,39.821,157.431
C04604=1034.059,-83.973,-81.090,167.995,39.820,157.431
C04605=1034.065,-83.689,-81.102,167.998,39.818,157.431
C04606=1034.071,-83.439,-81.113,168.001,39.817,157.431
C04607=1034.078,-83.189,-81.124,168.003,39.817,157.431
C04608=1034.084,-82.940,-81.134,168.006,39.816,157.431
C04609=1034.090,-82.690,-81.145,168.009,39.815,157.431
C04610=1034.096,-82.440,-81.156,168.011,39.814,157.431
C04611=1034.102,-82.190,-81.166,168.014,39.813,157.431
C04612=1034.108,-81.941,-81.177,168.017,39.812,157.431
C04613=1034.115,-81.691,-81.187,168.020,39.810,157.430
C04614=1034.121,-81.441,-81.198,168.023,39.809,157.430
C04615=1034.127,-81.191,-81.210,168.025,39.809,157.430
C04616=1034.134,-80.942,-81.220,168.027,39.808,157.430
C04617=1034.139,-80.693,-81.231,168.030,39.807,157.430
C04618=1034.146,-80.442,-81.242,168.033,39.806,157.430
C04619=1034.152,-80.193,-81.252,168.036,39.805,157.430
C04620=1034.159,-79.943,-81.263,168.038,39.804,157.430
///RCONF 1,0,0,0,0,0,0,0,0,0,0,0,0,0,0,0,0,0,0,0,0,0,0,0
C04621=1034.164,-79.694,-81.274,168.041,39.803,157.430
C04622=1034.170,-79.444,-81.285,168.044,39.802,157.430
C04623=1034.176,-79.194,-81.296,168.047,39.801,157.430
C04624=1034.182,-78.944,-81.307,168.049,39.801,157.430
C04625=1034.189,-78.695,-81.318,168.052,39.800,157.430
C04626=1034.195,-78.445,-81.329,168.054,39.799,157.430
C04627=1034.201,-78.195,-81.340,168.057,39.798,157.430
C04628=1034.207,-77.946,-81.352,168.059,39.798,157.430
C04629=1034.213,-77.696,-81.363,168.062,39.797,157.430
C04630=1034.219,-77.446,-81.374,168.065,39.796,157.430
C04631=1034.225,-77.197,-81.385,168.068,39.795,157.429
C04632=1034.231,-76.947,-81.396,168.070,39.794,157.429
C04633=1034.237,-76.697,-81.407,168.073,39.793,157.429
C04634=1034.243,-76.448,-81.418,168.076,39.792,157.429
C04635=1034.250,-76.198,-81.429,168.079,39.791,157.429
C04636=1034.256,-75.949,-81.440,168.081,39.790,157.429
C04637=1034.262,-75.699,-81.451,168.083,39.790,157.429
C04638=1034.268,-75.449,-81.462,168.086,39.789,157.429
C04639=1034.274,-75.199,-81.473,168.089,39.788,157.429
C04640=1034.281,-74.950,-81.485,168.091,39.788,157.429
C04641=1034.287,-74.700,-81.496,168.094,39.787,157.429
C04642=1034.293,-74.450,-81.507,168.097,39.786,157.429
C04643=1034.299,-74.200,-81.518,168.100,39.785,157.429
C04644=1034.305,-73.951,-81.529,168.102,39.784,157.429
C04645=1034.311,-73.702,-81.541,168.105,39.784,157.429
C04646=1034.317,-73.452,-81.552,168.108,39.783,157.429
C04647=1034.323,-73.202,-81.563,168.110,39.782,157.429
C04648=1034.329,-72.952,-81.575,168.113,39.781,157.429
C04649=1034.334,-72.703,-81.586,168.116,39.781,157.429
C04650=1034.341,-72.453,-81.598,168.119,39.780,157.429
C04651=1034.347,-72.204,-81.609,168.120,39.779,157.429
C04652=1034.353,-71.954,-81.620,168.123,39.779,157.429
C04653=1034.358,-71.704,-81.633,168.126,39.778,157.429
C04654=1034.365,-71.454,-81.644,168.128,39.777,157.429
C04655=1034.371,-71.205,-81.655,168.131,39.777,157.429
C04656=1034.377,-70.955,-81.667,168.134,39.776,157.429
C04657=1034.383,-70.706,-81.678,168.136,39.775,157.429
C04658=1034.390,-70.456,-81.689,168.139,39.774,157.428
C04659=1034.395,-70.206,-81.701,168.142,39.774,157.429
C04660=1034.401,-69.956,-81.712,168.144,39.773,157.428
C04661=1034.407,-69.707,-81.724,168.147,39.772,157.428
C04662=1034.413,-69.457,-81.735,168.150,39.772,157.429
C04663=1034.419,-69.207,-81.748,168.152,39.771,157.428
C04664=1034.425,-68.958,-81.758,168.155,39.770,157.428
C04665=1034.432,-68.708,-81.770,168.158,39.770,157.428
C04666=1034.438,-68.425,-81.783,168.161,39.769,157.428
C04667=1034.445,-68.143,-81.796,168.163,39.768,157.428
C04668=1034.452,-67.860,-81.809,168.166,39.767,157.428
C04669=1034.459,-67.577,-81.822,168.169,39.766,157.428
C04670=1034.465,-67.328,-81.834,168.172,39.766,157.428
C04671=1034.472,-67.078,-81.846,168.174,39.765,157.428
C04672=1034.477,-66.828,-81.858,168.177,39.764,157.428
C04673=1034.483,-66.578,-81.869,168.180,39.764,157.428
C04674=1034.489,-66.329,-81.881,168.182,39.763,157.428
C04675=1034.496,-66.079,-81.892,168.185,39.762,157.428
C04676=1034.502,-65.829,-81.904,168.188,39.762,157.428
C04677=1034.508,-65.580,-81.916,168.190,39.761,157.428
C04678=1034.514,-65.330,-81.927,168.193,39.760,157.428
C04679=1034.521,-65.081,-81.939,168.196,39.760,157.428
C04680=1034.526,-64.831,-81.950,168.198,39.759,157.428
C04681=1034.532,-64.581,-81.963,168.201,39.758,157.428
C04682=1034.539,-64.332,-81.975,168.204,39.758,157.428
C04683=1034.545,-64.082,-81.985,168.205,39.757,157.428
C04684=1034.551,-63.833,-81.997,168.208,39.756,157.428
C04685=1034.557,-63.583,-82.010,168.211,39.756,157.428
C04686=1034.563,-63.333,-82.021,168.213,39.755,157.428
C04687=1034.570,-63.084,-82.033,168.216,39.754,157.428
C04688=1034.575,-62.834,-82.045,168.219,39.754,157.428
C04689=1034.581,-62.584,-82.056,168.221,39.753,157.428
C04690=1034.588,-62.335,-82.068,168.224,39.752,157.428
C04691=1034.594,-62.085,-82.080,168.226,39.752,157.428
C04692=1034.600,-61.835,-82.092,168.229,39.751,157.428
C04693=1034.606,-61.586,-82.104,168.232,39.750,157.428
C04694=1034.613,-61.336,-82.116,168.234,39.750,157.428
C04695=1034.619,-61.087,-82.128,168.237,39.749,157.428
C04696=1034.625,-60.836,-82.139,168.240,39.748,157.428
C04697=1034.631,-60.587,-82.151,168.242,39.747,157.428
C04698=1034.638,-60.338,-82.163,168.245,39.747,157.428
C04699=1034.644,-60.088,-82.175,168.248,39.746,157.428
C04700=1034.650,-59.838,-82.187,168.249,39.745,157.428
C04701=1034.656,-59.589,-82.198,168.252,39.745,157.428
C04702=1034.663,-59.339,-82.210,168.255,39.744,157.428
C04703=1034.669,-59.089,-82.223,168.257,39.743,157.427
C04704=1034.675,-58.840,-82.235,168.260,39.743,157.428
C04705=1034.682,-58.590,-82.246,168.263,39.742,157.427
C04706=1034.687,-58.340,-82.258,168.265,39.741,157.427
C04707=1034.693,-58.091,-82.270,168.268,39.741,157.427
C04708=1034.700,-57.841,-82.282,168.271,39.740,157.427
C04709=1034.707,-57.592,-82.294,168.273,39.739,157.427
C04710=1034.713,-57.342,-82.307,168.276,39.739,157.427
C04711=1034.719,-57.093,-82.318,168.278,39.738,157.427
C04712=1034.725,-56.843,-82.330,168.281,39.737,157.427
C04713=1034.731,-56.593,-82.342,168.284,39.737,157.427
C04714=1034.738,-56.343,-82.354,168.286,39.736,157.427
C04715=1034.744,-56.094,-82.366,168.289,39.736,157.427
C04716=1034.750,-55.844,-82.379,168.292,39.735,157.427
C04717=1034.757,-55.594,-82.390,168.293,39.734,157.427
C04718=1034.763,-55.345,-82.402,168.296,39.734,157.427
C04719=1034.769,-55.095,-82.415,168.299,39.733,157.427
C04720=1034.775,-54.846,-82.427,168.301,39.732,157.427
C04721=1034.782,-54.596,-82.439,168.304,39.732,157.427
C04722=1034.789,-54.347,-82.451,168.306,39.731,157.427
C04723=1034.795,-54.097,-82.463,168.309,39.730,157.427
C04724=1034.801,-53.847,-82.475,168.312,39.730,157.427
C04725=1034.808,-53.598,-82.487,168.314,39.729,157.427
C04726=1034.814,-53.348,-82.500,168.317,39.728,157.427
C04727=1034.820,-53.098,-82.511,168.320,39.728,157.427
C04728=1034.827,-52.849,-82.523,168.322,39.727,157.427
C04729=1034.832,-52.600,-82.536,168.325,39.726,157.427
C04730=1034.839,-52.317,-82.549,168.328,39.726,157.427
C04731=1034.847,-52.036,-82.562,168.331,39.725,157.427
C04732=1034.854,-51.755,-82.577,168.334,39.724,157.427
C04733=1034.861,-51.473,-82.590,168.336,39.723,157.427
C04734=1034.868,-51.223,-82.602,168.338,39.723,157.427
C04735=1034.874,-50.974,-82.614,168.341,39.722,157.427
C04736=1034.880,-50.724,-82.627,168.344,39.721,157.427
C04737=1034.887,-50.475,-82.639,168.346,39.721,157.427
C04738=1034.893,-50.225,-82.652,168.349,39.720,157.427
C04739=1034.899,-49.975,-82.665,168.351,39.720,157.427
C04740=1034.906,-49.726,-82.676,168.354,39.720,157.427
C04741=1034.912,-49.476,-82.689,168.356,39.719,157.427
C04742=1034.918,-49.226,-82.702,168.359,39.719,157.427
C04743=1034.924,-48.977,-82.714,168.361,39.718,157.427
C04744=1034.930,-48.728,-82.726,168.364,39.718,157.427
C04745=1034.936,-48.478,-82.739,168.367,39.718,157.427
C04746=1034.942,-48.229,-82.752,168.369,39.717,157.427
C04747=1034.949,-47.979,-82.764,168.372,39.716,157.427
C04748=1034.954,-47.729,-82.777,168.374,39.716,157.427
C04749=1034.960,-47.479,-82.789,168.377,39.715,157.427
C04750=1034.967,-47.230,-82.802,168.379,39.715,157.427
C04751=1034.973,-46.980,-82.815,168.382,39.714,157.427
C04752=1034.979,-46.731,-82.827,168.384,39.714,157.427
C04753=1034.986,-46.482,-82.840,168.387,39.713,157.427
C04754=1034.992,-46.232,-82.852,168.389,39.713,157.427
C04755=1034.998,-45.982,-82.865,168.392,39.712,157.427
C04756=1035.004,-45.732,-82.877,168.394,39.712,157.427
C04757=1035.011,-45.483,-82.890,168.397,39.712,157.427
C04758=1035.017,-45.233,-82.903,168.400,39.711,157.427
C04759=1035.023,-44.984,-82.916,168.402,39.711,157.427
C04760=1035.029,-44.734,-82.928,168.405,39.710,157.427
C04761=1035.035,-44.484,-82.940,168.407,39.710,157.427
C04762=1035.042,-44.235,-82.954,168.410,39.709,157.427
C04763=1035.048,-43.985,-82.967,168.412,39.708,157.427
C04764=1035.055,-43.735,-82.979,168.415,39.708,157.427
C04765=1035.061,-43.486,-82.992,168.416,39.707,157.427
C04766=1035.067,-43.236,-83.004,168.420,39.707,157.427
C04767=1035.073,-42.987,-83.018,168.422,39.707,157.427
C04768=1035.080,-42.737,-83.030,168.424,39.706,157.427
C04769=1035.086,-42.487,-83.042,168.426,39.706,157.427
C04770=1035.092,-42.238,-83.055,168.429,39.705,157.427
C04771=1035.098,-41.988,-83.068,168.431,39.705,157.427
C04772=1035.105,-41.739,-83.081,168.434,39.705,157.427
C04773=1035.111,-41.489,-83.093,168.436,39.704,157.427
C04774=1035.117,-41.240,-83.107,168.439,39.704,157.427
C04775=1035.123,-40.989,-83.119,168.441,39.703,157.427
C04776=1035.130,-40.740,-83.132,168.444,39.702,157.427
C04777=1035.136,-40.490,-83.145,168.447,39.702,157.427
C04778=1035.142,-40.241,-83.158,168.449,39.701,157.427
C04779=1035.148,-39.991,-83.171,168.452,39.701,157.427
C04780=1035.155,-39.742,-83.184,168.454,39.700,157.427
C04781=1035.161,-39.492,-83.196,168.457,39.700,157.427
C04782=1035.168,-39.242,-83.209,168.459,39.699,157.427
C04783=1035.174,-38.993,-83.222,168.462,39.699,157.427
C04784=1035.180,-38.743,-83.235,168.464,39.699,157.427
C04785=1035.186,-38.494,-83.248,168.467,39.698,157.427
C04786=1035.192,-38.244,-83.261,168.469,39.698,157.427
C04787=1035.199,-37.995,-83.274,168.471,39.698,157.427
C04788=1035.205,-37.746,-83.288,168.474,39.697,157.427
C04789=1035.211,-37.495,-83.300,168.476,39.697,157.427
C04790=1035.217,-37.246,-83.314,168.479,39.696,157.427
C04791=1035.224,-36.997,-83.327,168.481,39.696,157.427
C04792=1035.230,-36.747,-83.340,168.484,39.696,157.427
C04793=1035.236,-36.497,-83.353,168.486,39.695,157.427
C04794=1035.243,-36.216,-83.367,168.489,39.695,157.427
C04795=1035.251,-35.935,-83.382,168.492,39.695,157.427
C04796=1035.257,-35.654,-83.397,168.495,39.694,157.427
C04797=1035.264,-35.373,-83.411,168.497,39.693,157.427
C04798=1035.270,-35.123,-83.425,168.500,39.693,157.427
C04799=1035.277,-34.874,-83.438,168.502,39.693,157.427
C04800=1035.283,-34.624,-83.452,168.505,39.693,157.428
C04801=1035.289,-34.374,-83.464,168.507,39.692,157.427
C04802=1035.296,-34.125,-83.477,168.510,39.692,157.428
C04803=1035.302,-33.876,-83.491,168.512,39.692,157.428
C04804=1035.308,-33.627,-83.504,168.515,39.691,157.428
C04805=1035.315,-33.377,-83.518,168.517,39.691,157.428
C04806=1035.321,-33.127,-83.530,168.519,39.690,157.428
C04807=1035.327,-32.877,-83.543,168.522,39.690,157.428
C04808=1035.333,-32.628,-83.557,168.524,39.690,157.428
C04809=1035.339,-32.378,-83.571,168.527,39.689,157.428
C04810=1035.345,-32.129,-83.584,168.529,39.689,157.428
C04811=1035.351,-31.879,-83.597,168.532,39.689,157.428
C04812=1035.358,-31.630,-83.610,168.534,39.688,157.428
C04813=1035.364,-31.380,-83.624,168.537,39.688,157.428
C04814=1035.371,-31.130,-83.637,168.539,39.687,157.428
C04815=1035.377,-30.881,-83.650,168.541,39.687,157.428
C04816=1035.384,-30.631,-83.664,168.544,39.686,157.428
C04817=1035.390,-30.382,-83.677,168.546,39.686,157.428
C04818=1035.396,-30.132,-83.690,168.549,39.686,157.428
C04819=1035.403,-29.882,-83.703,168.551,39.686,157.428
C04820=1035.409,-29.633,-83.717,168.554,39.685,157.428
C04821=1035.415,-29.383,-83.730,168.556,39.685,157.428
C04822=1035.422,-29.133,-83.744,168.559,39.684,157.428
C04823=1035.428,-28.884,-83.757,168.561,39.684,157.428
C04824=1035.434,-28.635,-83.770,168.563,39.683,157.428
C04825=1035.441,-28.385,-83.784,168.566,39.683,157.428
C04826=1035.447,-28.136,-83.797,168.568,39.683,157.428
C04827=1035.453,-27.886,-83.811,168.571,39.683,157.428
C04828=1035.460,-27.636,-83.824,168.573,39.682,157.428
C04829=1035.466,-27.387,-83.838,168.576,39.682,157.428
C04830=1035.472,-27.138,-83.851,168.578,39.682,157.428
C04831=1035.479,-26.888,-83.865,168.580,39.681,157.428
C04832=1035.485,-26.638,-83.878,168.583,39.681,157.428
C04833=1035.490,-26.389,-83.892,168.585,39.680,157.428
C04834=1035.497,-26.139,-83.905,168.587,39.680,157.428
C04835=1035.504,-25.890,-83.919,168.590,39.680,157.428
C04836=1035.509,-25.640,-83.933,168.592,39.680,157.428
C04837=1035.516,-25.390,-83.946,168.595,39.679,157.428
C04838=1035.522,-25.141,-83.959,168.597,39.679,157.428
C04839=1035.528,-24.891,-83.974,168.599,39.679,157.428
C04840=1035.535,-24.642,-83.988,168.602,39.679,157.429
C04841=1035.541,-24.393,-84.001,168.604,39.679,157.429
C04842=1035.547,-24.142,-84.015,168.607,39.679,157.429
C04843=1035.553,-23.893,-84.028,168.609,39.678,157.429
C04844=1035.559,-23.644,-84.042,168.611,39.678,157.429
C04845=1035.565,-23.394,-84.056,168.614,39.677,157.429
C04846=1035.572,-23.145,-84.070,168.616,39.677,157.429
C04847=1035.579,-22.895,-84.084,168.618,39.677,157.429
C04848=1035.584,-22.645,-84.097,168.621,39.677,157.429
C04849=1035.591,-22.395,-84.111,168.623,39.677,157.429
C04850=1035.597,-22.146,-84.124,168.625,39.676,157.429
C04851=1035.603,-21.897,-84.139,168.628,39.676,157.429
C04852=1035.610,-21.647,-84.153,168.630,39.675,157.429
C04853=1035.616,-21.398,-84.166,168.633,39.675,157.429
C04854=1035.622,-21.148,-84.180,168.635,39.675,157.429
C04855=1035.628,-20.898,-84.193,168.637,39.675,157.429
C04856=1035.635,-20.649,-84.208,168.640,39.674,157.429
C04857=1035.641,-20.399,-84.222,168.642,39.674,157.429
C04858=1035.648,-20.117,-84.237,168.645,39.674,157.429
C04859=1035.655,-19.836,-84.253,168.647,39.674,157.429
C04860=1035.663,-19.554,-84.269,168.650,39.673,157.429
C04861=1035.669,-19.272,-84.284,168.653,39.673,157.429
C04862=1035.676,-19.023,-84.298,168.655,39.673,157.429
C04863=1035.683,-18.774,-84.311,168.657,39.672,157.429
C04864=1035.689,-18.523,-84.326,168.660,39.672,157.429
C04865=1035.695,-18.274,-84.339,168.662,39.672,157.429
C04866=1035.701,-18.025,-84.354,168.665,39.672,157.429
C04867=1035.708,-17.775,-84.367,168.667,39.672,157.430
C04868=1035.714,-17.525,-84.381,168.669,39.671,157.429
C04869=1035.721,-17.276,-84.396,168.672,39.671,157.430
C04870=1035.727,-17.026,-84.409,168.674,39.670,157.430
C04871=1035.734,-16.777,-84.423,168.676,39.670,157.430
C04872=1035.739,-16.527,-84.437,168.679,39.670,157.430
C04873=1035.746,-16.278,-84.451,168.681,39.670,157.430
C04874=1035.752,-16.029,-84.465,168.683,39.670,157.430
C04875=1035.759,-15.779,-84.479,168.686,39.669,157.430
C04876=1035.765,-15.530,-84.493,168.688,39.669,157.430
C04877=1035.771,-15.280,-84.507,168.690,39.668,157.430
C04878=1035.778,-15.030,-84.521,168.693,39.668,157.430
C04879=1035.784,-14.781,-84.535,168.695,39.668,157.430
C04880=1035.790,-14.530,-84.550,168.697,39.668,157.430
C04881=1035.797,-14.282,-84.564,168.700,39.668,157.430
C04882=1035.803,-14.032,-84.579,168.702,39.667,157.430
C04883=1035.809,-13.783,-84.593,168.704,39.667,157.430
C04884=1035.816,-13.533,-84.607,168.706,39.667,157.430
C04885=1035.821,-13.284,-84.621,168.709,39.667,157.430
C04886=1035.828,-13.034,-84.635,168.711,39.667,157.430
C04887=1035.834,-12.785,-84.649,168.713,39.667,157.430
C04888=1035.840,-12.535,-84.664,168.716,39.667,157.430
C04889=1035.847,-12.285,-84.678,168.718,39.667,157.430
C04890=1035.853,-12.036,-84.692,168.720,39.667,157.431
C04891=1035.859,-11.787,-84.707,168.723,39.666,157.431
C04892=1035.865,-11.537,-84.720,168.725,39.666,157.431
C04893=1035.872,-11.288,-84.735,168.728,39.666,157.431
C04894=1035.878,-11.037,-84.749,168.730,39.666,157.431
C04895=1035.884,-10.789,-84.763,168.733,39.666,157.431
C04896=1035.891,-10.539,-84.778,168.735,39.665,157.431
C04897=1035.897,-10.289,-84.792,168.737,39.665,157.431
C04898=1035.903,-10.040,-84.807,168.740,39.665,157.431
C04899=1035.909,-9.790,-84.821,168.742,39.665,157.431
C04900=1035.916,-9.541,-84.835,168.744,39.665,157.431
C04901=1035.922,-9.292,-84.850,168.746,39.665,157.431
C04902=1035.928,-9.041,-84.864,168.749,39.664,157.431
C04903=1035.935,-8.793,-84.878,168.751,39.664,157.431
C04904=1035.941,-8.543,-84.893,168.753,39.664,157.431
C04905=1035.948,-8.293,-84.908,168.756,39.664,157.431
C04906=1035.954,-8.044,-84.921,168.758,39.664,157.431
C04907=1035.960,-7.794,-84.936,168.760,39.663,157.431
C04908=1035.967,-7.545,-84.951,168.762,39.663,157.431
C04909=1035.973,-7.295,-84.964,168.765,39.663,157.431
C04910=1035.979,-7.046,-84.979,168.767,39.663,157.432
C04911=1035.986,-6.796,-84.994,168.769,39.663,157.432
C04912=1035.993,-6.547,-85.009,168.772,39.662,157.432
C04913=1035.998,-6.297,-85.022,168.774,39.662,157.432
C04914=1036.005,-6.048,-85.037,168.776,39.662,157.432
C04915=1036.012,-5.798,-85.052,168.778,39.662,157.432
C04916=1036.017,-5.549,-85.066,168.781,39.661,157.432
C04917=1036.024,-5.299,-85.081,168.783,39.661,157.432
C04918=1036.031,-5.050,-85.095,168.785,39.661,157.432
C04919=1036.037,-4.800,-85.110,168.787,39.661,157.432
C04920=1036.043,-4.551,-85.124,168.790,39.660,157.432
C04921=1036.050,-4.302,-85.139,168.792,39.660,157.432
C04922=1036.057,-4.018,-85.155,168.795,39.660,157.432
C04923=1036.064,-3.735,-85.171,168.797,39.660,157.432
C04924=1036.071,-3.450,-85.189,168.800,39.660,157.432
C04925=1036.078,-3.167,-85.206,168.802,39.660,157.432
C04926=1036.084,-2.918,-85.220,168.804,39.660,157.432
C04927=1036.091,-2.669,-85.235,168.807,39.660,157.432
C04928=1036.097,-2.419,-85.250,168.809,39.659,157.432
C04929=1036.103,-2.170,-85.265,168.811,39.659,157.432
C04930=1036.109,-1.920,-85.280,168.813,39.660,157.433
C04931=1036.115,-1.670,-85.294,168.816,39.660,157.433
C04932=1036.122,-1.421,-85.309,168.819,39.659,157.433
C04933=1036.127,-1.172,-85.324,168.821,39.659,157.433
C04934=1036.134,-0.922,-85.339,168.823,39.659,157.433
C04935=1036.140,-0.672,-85.354,168.825,39.659,157.433
C04936=1036.147,-0.423,-85.368,168.827,39.659,157.433
C04937=1036.153,-0.174,-85.384,168.830,39.659,157.433
C04938=1036.159,0.075,-85.399,168.832,39.659,157.433
C04939=1036.165,0.325,-85.414,168.834,39.659,157.433
C04940=1036.172,0.575,-85.429,168.836,39.659,157.433
C04941=1036.178,0.824,-85.444,168.839,39.659,157.433
C04942=1036.184,1.073,-85.458,168.841,39.659,157.433
C04943=1036.190,1.323,-85.473,168.843,39.659,157.433
C04944=1036.197,1.573,-85.488,168.845,39.658,157.434
C04945=1036.203,1.822,-85.503,168.847,39.658,157.434
C04946=1036.209,2.072,-85.518,168.850,39.658,157.434
C04947=1036.215,2.321,-85.532,168.852,39.658,157.434
C04948=1036.222,2.571,-85.547,168.854,39.658,157.434
C04949=1036.228,2.820,-85.562,168.856,39.658,157.434
C04950=1036.234,3.070,-85.577,168.858,39.658,157.434
C04951=1036.241,3.319,-85.593,168.861,39.658,157.434
C04952=1036.247,3.568,-85.608,168.863,39.658,157.434
C04953=1036.253,3.817,-85.623,168.865,39.657,157.434
C04954=1036.260,4.067,-85.637,168.868,39.658,157.434
C04955=1036.266,4.317,-85.652,168.870,39.658,157.434
C04956=1036.272,4.566,-85.667,168.872,39.658,157.434
C04957=1036.278,4.816,-85.684,168.875,39.657,157.434
C04958=1036.285,5.065,-85.699,168.877,39.657,157.434
C04959=1036.291,5.315,-85.713,168.879,39.657,157.434
C04960=1036.297,5.564,-85.728,168.881,39.657,157.434
C04961=1036.303,5.814,-85.743,168.883,39.657,157.435
C04962=1036.310,6.063,-85.759,168.886,39.657,157.435
C04963=1036.316,6.312,-85.774,168.888,39.657,157.435
C04964=1036.323,6.562,-85.789,168.890,39.657,157.435
C04965=1036.329,6.812,-85.804,168.892,39.657,157.435
C04966=1036.336,7.061,-85.818,168.894,39.656,157.435
C04967=1036.342,7.310,-85.834,168.897,39.656,157.435
C04968=1036.349,7.560,-85.849,168.899,39.656,157.435
C04969=1036.355,7.810,-85.864,168.901,39.657,157.435
C04970=1036.361,8.059,-85.879,168.903,39.656,157.435
C04971=1036.367,8.308,-85.894,168.905,39.656,157.435
C04972=1036.374,8.557,-85.909,168.908,39.656,157.435
C04973=1036.380,8.807,-85.924,168.910,39.656,157.435
C04974=1036.386,9.056,-85.940,168.912,39.656,157.435
C04975=1036.393,9.306,-85.955,168.914,39.656,157.435
C04976=1036.399,9.556,-85.970,168.916,39.655,157.435
C04977=1036.406,9.805,-85.986,168.918,39.655,157.436
C04978=1036.412,10.054,-86.001,168.921,39.656,157.436
C04979=1036.418,10.304,-86.016,168.923,39.655,157.436
C04980=1036.425,10.553,-86.032,168.926,39.655,157.436
C04981=1036.431,10.803,-86.046,168.928,39.655,157.436
C04982=1036.438,11.052,-86.061,168.930,39.655,157.436
C04983=1036.445,11.301,-86.077,168.933,39.655,157.436
C04984=1036.451,11.551,-86.092,168.935,39.655,157.436
C04985=1036.457,11.801,-86.107,168.937,39.654,157.436
C04986=1036.464,12.067,-86.124,168.939,39.654,157.436
C04987=1036.471,12.334,-86.140,168.942,39.655,157.436
C04988=1036.478,12.601,-86.157,168.944,39.654,157.436
C04989=1036.485,12.868,-86.173,168.946,39.654,157.436
C04990=1036.493,13.192,-86.193,168.949,39.654,157.436
C04991=1036.499,13.441,-86.208,168.951,39.654,157.436
C04992=1036.506,13.690,-86.224,168.953,39.654,157.436
C04993=1036.513,13.940,-86.239,168.956,39.653,157.437
C04994=1036.519,14.189,-86.254,168.958,39.653,157.437
C04995=1036.525,14.439,-86.270,168.960,39.654,157.437
C04996=1036.532,14.688,-86.286,168.962,39.654,157.437
C04997=1036.538,14.938,-86.301,168.964,39.653,157.437
C04998=1036.544,15.187,-86.317,168.966,39.653,157.437
C04999=1036.550,15.437,-86.332,168.968,39.654,157.437
C05000=1036.557,15.686,-86.347,168.970,39.654,157.437
C05001=1036.563,15.935,-86.364,168.973,39.653,157.437
C05002=1036.569,16.185,-86.379,168.975,39.653,157.437
C05003=1036.575,16.434,-86.395,168.978,39.654,157.437
C05004=1036.582,16.684,-86.410,168.980,39.654,157.437
C05005=1036.588,16.933,-86.426,168.982,39.653,157.437
C05006=1036.594,17.183,-86.441,168.984,39.653,157.437
C05007=1036.601,17.432,-86.457,168.986,39.653,157.438
C05008=1036.607,17.681,-86.472,168.989,39.653,157.438
C05009=1036.613,17.931,-86.488,168.991,39.653,157.438
C05010=1036.620,18.180,-86.504,168.993,39.653,157.438
C05011=1036.626,18.429,-86.519,168.995,39.653,157.438
C05012=1036.633,18.680,-86.535,168.997,39.653,157.438
C05013=1036.639,18.929,-86.551,168.999,39.653,157.438
C05014=1036.645,19.178,-86.567,169.001,39.653,157.438
C05015=1036.652,19.428,-86.582,169.003,39.653,157.438
C05016=1036.658,19.677,-86.598,169.006,39.653,157.438
C05017=1036.664,19.926,-86.614,169.008,39.653,157.438
C05018=1036.671,20.176,-86.629,169.010,39.653,157.438
C05019=1036.677,20.425,-86.645,169.012,39.653,157.438
C05020=1036.683,20.674,-86.661,169.014,39.653,157.438
C05021=1036.689,20.923,-86.677,169.016,39.653,157.439
C05022=1036.696,21.174,-86.692,169.018,39.653,157.439
C05023=1036.702,21.423,-86.709,169.020,39.653,157.439
C05024=1036.709,21.672,-86.724,169.023,39.653,157.439
C05025=1036.715,21.921,-86.741,169.025,39.653,157.439
C05026=1036.721,22.171,-86.755,169.028,39.653,157.439
C05027=1036.727,22.420,-86.772,169.030,39.653,157.439
C05028=1036.734,22.669,-86.787,169.032,39.653,157.439
C05029=1036.740,22.919,-86.804,169.034,39.653,157.439
C05030=1036.747,23.169,-86.820,169.036,39.653,157.439
C05031=1036.753,23.419,-86.835,169.038,39.653,157.439
C05032=1036.759,23.668,-86.851,169.040,39.653,157.439
C05033=1036.765,23.917,-86.867,169.042,39.653,157.440
C05034=1036.772,24.166,-86.883,169.044,39.653,157.440
C05035=1036.778,24.415,-86.899,169.046,39.653,157.440
C05036=1036.785,24.664,-86.915,169.048,39.653,157.440
C05037=1036.791,24.914,-86.931,169.051,39.653,157.440
C05038=1036.797,25.164,-86.947,169.053,39.653,157.440
C05039=1036.804,25.413,-86.963,169.055,39.653,157.440
C05040=1036.810,25.663,-86.979,169.057,39.653,157.440
C05041=1036.816,25.912,-86.994,169.059,39.653,157.440
C05042=1036.823,26.162,-87.011,169.062,39.653,157.440
C05043=1036.829,26.411,-87.027,169.064,39.653,157.440
C05044=1036.835,26.660,-87.043,169.066,39.653,157.440
C05045=1036.842,26.909,-87.059,169.068,39.653,157.440
C05046=1036.848,27.159,-87.075,169.070,39.653,157.440
C05047=1036.855,27.409,-87.092,169.072,39.653,157.441
C05048=1036.861,27.658,-87.107,169.075,39.653,157.441
C05049=1036.867,27.907,-87.123,169.077,39.653,157.441
C05050=1036.874,28.194,-87.141,169.079,39.653,157.441
C05051=1036.882,28.480,-87.160,169.081,39.653,157.441
C05052=1036.890,28.767,-87.179,169.084,39.653,157.441
C05053=1036.896,29.054,-87.198,169.086,39.653,157.441
C05054=1036.903,29.303,-87.213,169.088,39.653,157.441
C05055=1036.909,29.553,-87.229,169.090,39.654,157.441
C05056=1036.915,29.802,-87.246,169.092,39.654,157.441
C05057=1036.921,30.052,-87.262,169.094,39.653,157.441
C05058=1036.928,30.300,-87.279,169.097,39.654,157.442
C05059=1036.934,30.550,-87.295,169.099,39.654,157.442
C05060=1036.940,30.799,-87.311,169.102,39.653,157.442
C05061=1036.947,31.049,-87.328,169.104,39.654,157.442
C05062=1036.953,31.299,-87.344,169.106,39.654,157.442
C05063=1036.959,31.548,-87.360,169.108,39.654,157.442
C05064=1036.965,31.797,-87.376,169.110,39.654,157.442
C05065=1036.972,32.047,-87.393,169.112,39.654,157.442
C05066=1036.978,32.296,-87.409,169.114,39.654,157.442
C05067=1036.985,32.545,-87.425,169.116,39.654,157.442
C05068=1036.991,32.794,-87.442,169.118,39.654,157.442
C05069=1036.997,33.044,-87.458,169.120,39.654,157.442
C05070=1037.003,33.294,-87.474,169.122,39.654,157.443
C05071=1037.010,33.543,-87.490,169.124,39.654,157.443
C05072=1037.016,33.793,-87.507,169.126,39.654,157.443
C05073=1037.023,34.041,-87.524,169.129,39.655,157.443
C05074=1037.029,34.291,-87.540,169.131,39.654,157.443
C05075=1037.035,34.541,-87.557,169.133,39.654,157.443
C05076=1037.042,34.790,-87.572,169.135,39.655,157.443
C05077=1037.048,35.039,-87.589,169.138,39.654,157.443
C05078=1037.055,35.289,-87.606,169.140,39.654,157.443
C05079=1037.061,35.538,-87.622,169.142,39.655,157.443
C05080=1037.067,35.787,-87.638,169.144,39.655,157.443
C05081=1037.074,36.037,-87.654,169.146,39.654,157.443
C05082=1037.080,36.286,-87.671,169.148,39.655,157.444
C05083=1037.086,36.535,-87.688,169.150,39.655,157.444
C05084=1037.093,36.785,-87.704,169.152,39.655,157.444
C05085=1037.099,37.034,-87.720,169.154,39.654,157.444
C05086=1037.106,37.283,-87.737,169.156,39.655,157.444
C05087=1037.112,37.533,-87.753,169.158,39.655,157.444
C05088=1037.118,37.782,-87.770,169.161,39.655,157.444
C05089=1037.124,38.031,-87.787,169.163,39.655,157.444
C05090=1037.131,38.281,-87.803,169.165,39.655,157.444
C05091=1037.137,38.530,-87.820,169.167,39.655,157.444
C05092=1037.143,38.779,-87.837,169.169,39.655,157.444
C05093=1037.150,39.029,-87.853,169.171,39.656,157.445
C05094=1037.156,39.279,-87.869,169.173,39.656,157.445
C05095=1037.163,39.528,-87.887,169.175,39.656,157.445
C05096=1037.168,39.777,-87.903,169.177,39.656,157.445
C05097=1037.174,40.026,-87.921,169.179,39.656,157.445
C05098=1037.181,40.276,-87.937,169.181,39.656,157.445
C05099=1037.186,40.526,-87.953,169.183,39.656,157.445
C05100=1037.193,40.774,-87.970,169.185,39.657,157.445
C05101=1037.199,41.025,-87.987,169.187,39.656,157.445
C05102=1037.206,41.273,-88.004,169.189,39.656,157.445
C05103=1037.212,41.523,-88.021,169.192,39.657,157.446
C05104=1037.218,41.772,-88.038,169.194,39.656,157.446
C05105=1037.224,42.021,-88.054,169.196,39.657,157.446
C05106=1037.231,42.271,-88.071,169.198,39.657,157.446
C05107=1037.237,42.520,-88.088,169.200,39.657,157.446
C05108=1037.244,42.770,-88.105,169.202,39.657,157.446
C05109=1037.250,43.019,-88.121,169.204,39.657,157.446
C05110=1037.256,43.268,-88.138,169.206,39.657,157.446
C05111=1037.263,43.518,-88.155,169.208,39.657,157.446
C05112=1037.268,43.767,-88.172,169.210,39.658,157.446
C05113=1037.275,44.017,-88.189,169.212,39.658,157.446
C05114=1037.282,44.303,-88.209,169.216,39.658,157.447
C05115=1037.288,44.589,-88.228,169.218,39.658,157.447
C05116=1037.296,44.876,-88.247,169.220,39.658,157.447
C05117=1037.303,45.162,-88.267,169.223,39.659,157.447
C05118=1037.309,45.413,-88.284,169.225,39.659,157.447
C05119=1037.315,45.661,-88.301,169.226,39.659,157.447
C05120=1037.322,45.910,-88.318,169.228,39.659,157.447
C05121=1037.328,46.160,-88.335,169.230,39.659,157.447
C05122=1037.334,46.409,-88.352,169.232,39.659,157.447
C05123=1037.341,46.659,-88.370,169.234,39.660,157.448
C05124=1037.347,46.908,-88.386,169.236,39.660,157.448
C05125=1037.353,47.158,-88.404,169.239,39.660,157.448
C05126=1037.359,47.406,-88.421,169.241,39.660,157.448
C05127=1037.365,47.656,-88.437,169.243,39.660,157.448
C05128=1037.371,47.905,-88.455,169.245,39.660,157.448
C05129=1037.377,48.154,-88.472,169.247,39.661,157.448
C05130=1037.384,48.404,-88.489,169.249,39.661,157.448
C05131=1037.390,48.653,-88.506,169.251,39.661,157.448
C05132=1037.396,48.903,-88.524,169.253,39.661,157.449
C05133=1037.402,49.151,-88.541,169.255,39.661,157.449
C05134=1037.409,49.401,-88.557,169.257,39.661,157.449
C05135=1037.415,49.651,-88.575,169.259,39.662,157.449
C05136=1037.421,49.900,-88.592,169.261,39.661,157.449
C05137=1037.428,50.149,-88.609,169.264,39.662,157.449
C05138=1037.434,50.398,-88.627,169.266,39.662,157.449
C05139=1037.440,50.648,-88.643,169.268,39.662,157.449
C05140=1037.447,50.897,-88.661,169.270,39.662,157.449
C05141=1037.452,51.146,-88.678,169.272,39.663,157.450
C05142=1037.459,51.396,-88.695,169.274,39.662,157.450
C05143=1037.465,51.645,-88.712,169.276,39.663,157.450
C05144=1037.471,51.895,-88.730,169.278,39.663,157.450
C05145=1037.478,52.144,-88.747,169.280,39.663,157.450
C05146=1037.484,52.393,-88.764,169.282,39.663,157.450
C05147=1037.490,52.643,-88.782,169.284,39.663,157.450
C05148=1037.497,52.891,-88.799,169.286,39.663,157.450
C05149=1037.503,53.141,-88.816,169.288,39.663,157.450
C05150=1037.509,53.390,-88.833,169.291,39.664,157.450
C05151=1037.515,53.640,-88.850,169.293,39.664,157.450
C05152=1037.522,53.889,-88.867,169.295,39.664,157.451
C05153=1037.528,54.138,-88.885,169.297,39.664,157.451
C05154=1037.535,54.388,-88.903,169.299,39.664,157.451
C05155=1037.541,54.637,-88.920,169.301,39.664,157.451
C05156=1037.547,54.886,-88.938,169.303,39.665,157.451
C05157=1037.553,55.135,-88.955,169.305,39.664,157.451
C05158=1037.560,55.385,-88.971,169.307,39.664,157.451
C05159=1037.566,55.635,-88.989,169.309,39.665,157.451
C05160=1037.572,55.884,-89.006,169.311,39.665,157.451
C05161=1037.579,56.133,-89.023,169.313,39.665,157.451
C05162=1037.585,56.382,-89.041,169.315,39.665,157.451
C05163=1037.591,56.631,-89.058,169.318,39.665,157.452
C05164=1037.598,56.881,-89.076,169.320,39.665,157.452
C05165=1037.604,57.130,-89.093,169.322,39.665,157.452
C05166=1037.611,57.379,-89.111,169.324,39.666,157.452
C05167=1037.617,57.629,-89.128,169.326,39.665,157.452
C05168=1037.623,57.878,-89.145,169.328,39.666,157.452
C05169=1037.630,58.127,-89.163,169.330,39.666,157.452
C05170=1037.636,58.377,-89.181,169.332,39.666,157.452
C05171=1037.642,58.626,-89.198,169.334,39.666,157.452
C05172=1037.649,58.875,-89.215,169.336,39.666,157.452
C05173=1037.655,59.125,-89.233,169.338,39.666,157.453
C05174=1037.662,59.374,-89.250,169.340,39.666,157.453
C05175=1037.668,59.623,-89.268,169.343,39.667,157.453
C05176=1037.675,59.873,-89.285,169.345,39.666,157.453
C05177=1037.681,60.121,-89.302,169.347,39.666,157.453
C05178=1037.688,60.408,-89.323,169.349,39.667,157.453
C05179=1037.695,60.694,-89.342,169.352,39.667,157.453
C05180=1037.703,60.981,-89.363,169.354,39.667,157.453
C05181=1037.710,61.267,-89.383,169.356,39.667,157.453
C05182=1037.717,61.516,-89.400,169.358,39.667,157.453
C05183=1037.723,61.765,-89.419,169.360,39.667,157.454
C05184=1037.730,62.015,-89.436,169.362,39.667,157.454
C05185=1037.736,62.263,-89.453,169.364,39.667,157.454
C05186=1037.742,62.513,-89.471,169.366,39.667,157.454
C05187=1037.749,62.763,-89.488,169.368,39.668,157.454
C05188=1037.755,63.012,-89.506,169.370,39.668,157.454
C05189=1037.762,63.261,-89.523,169.372,39.667,157.454
C05190=1037.768,63.510,-89.541,169.375,39.668,157.454
C05191=1037.775,63.760,-89.559,169.377,39.668,157.454
C05192=1037.782,64.009,-89.577,169.379,39.668,157.454
C05193=1037.787,64.258,-89.594,169.381,39.668,157.454
C05194=1037.793,64.508,-89.612,169.383,39.669,157.455
C05195=1037.800,64.757,-89.629,169.385,39.668,157.455
C05196=1037.807,65.006,-89.648,169.387,39.669,157.455
C05197=1037.812,65.255,-89.666,169.389,39.669,157.455
C05198=1037.819,65.505,-89.683,169.391,39.669,157.455
C05199=1037.825,65.754,-89.702,169.393,39.669,157.455
C05200=1037.831,66.003,-89.719,169.395,39.669,157.455
C05201=1037.838,66.252,-89.736,169.397,39.669,157.455
C05202=1037.844,66.502,-89.754,169.400,39.670,157.455
C05203=1037.850,66.751,-89.773,169.402,39.670,157.455
C05204=1037.857,67.001,-89.790,169.404,39.670,157.456
C05205=1037.863,67.250,-89.808,169.406,39.670,157.456
C05206=1037.869,67.499,-89.827,169.408,39.670,157.456
C05207=1037.875,67.749,-89.845,169.410,39.670,157.456
C05208=1037.882,67.998,-89.862,169.412,39.671,157.456
C05209=1037.888,68.246,-89.880,169.414,39.671,157.456
C05210=1037.894,68.496,-89.898,169.416,39.671,157.456
C05211=1037.900,68.746,-89.916,169.418,39.671,157.456
C05212=1037.907,68.995,-89.934,169.419,39.671,157.456
C05213=1037.913,69.244,-89.952,169.422,39.672,157.457
C05214=1037.919,69.493,-89.970,169.424,39.672,157.457
C05215=1037.925,69.743,-89.988,169.426,39.672,157.457
C05216=1037.932,69.992,-90.007,169.428,39.672,157.457
C05217=1037.939,70.241,-90.024,169.430,39.672,157.457
C05218=1037.944,70.490,-90.042,169.432,39.672,157.457
C05219=1037.951,70.739,-90.060,169.434,39.673,157.457
C05220=1037.957,70.989,-90.078,169.436,39.673,157.457
C05221=1037.963,71.238,-90.097,169.438,39.673,157.457
C05222=1037.969,71.488,-90.115,169.440,39.674,157.458
C05223=1037.975,71.736,-90.133,169.443,39.673,157.458
C05224=1037.982,71.986,-90.151,169.445,39.674,157.458
C05225=1037.988,72.235,-90.169,169.447,39.674,157.458
C05226=1037.995,72.485,-90.187,169.449,39.674,157.458
C05227=1038.001,72.734,-90.206,169.451,39.675,157.458
C05228=1038.007,72.984,-90.224,169.453,39.675,157.458
C05229=1038.013,73.232,-90.242,169.455,39.675,157.458
C05230=1038.019,73.482,-90.260,169.457,39.675,157.458
C05231=1038.026,73.731,-90.279,169.459,39.675,157.459
C05232=1038.032,73.980,-90.297,169.461,39.675,157.459
C05233=1038.039,74.229,-90.315,169.463,39.676,157.459
C05234=1038.045,74.478,-90.333,169.466,39.676,157.459
C05235=1038.051,74.727,-90.351,169.467,39.676,157.459
C05236=1038.057,74.977,-90.369,169.469,39.676,157.459
C05237=1038.064,75.226,-90.388,169.471,39.676,157.459
C05238=1038.070,75.475,-90.406,169.473,39.677,157.459
C05239=1038.076,75.725,-90.425,169.475,39.677,157.459
C05240=1038.082,75.974,-90.443,169.477,39.677,157.460
C05241=1038.089,76.223,-90.461,169.479,39.678,157.460
C05242=1038.096,76.509,-90.482,169.482,39.677,157.460
C05243=1038.103,76.795,-90.504,169.484,39.678,157.460
C05244=1038.111,77.082,-90.524,169.486,39.678,157.460
C05245=1038.117,77.367,-90.545,169.489,39.678,157.460
C05246=1038.124,77.616,-90.564,169.491,39.679,157.460
C05247=1038.130,77.866,-90.582,169.493,39.678,157.460
C05248=1038.136,78.115,-90.600,169.495,39.679,157.461
C05249=1038.143,78.364,-90.619,169.497,39.679,157.461
C05250=1038.149,78.614,-90.638,169.499,39.679,157.461
C05251=1038.155,78.863,-90.656,169.501,39.680,157.461
C05252=1038.161,79.112,-90.674,169.503,39.680,157.461
C05253=1038.167,79.361,-90.693,169.505,39.680,157.461
C05254=1038.173,79.610,-90.712,169.508,39.680,157.461
C05255=1038.180,79.859,-90.730,169.510,39.681,157.461
C05256=1038.186,80.109,-90.748,169.512,39.681,157.462
C05257=1038.192,80.358,-90.767,169.514,39.681,157.462
C05258=1038.198,80.607,-90.786,169.515,39.682,157.462
C05259=1038.204,80.857,-90.805,169.517,39.682,157.462
C05260=1038.211,81.106,-90.824,169.519,39.682,157.462
C05261=1038.217,81.355,-90.842,169.521,39.683,157.462
C05262=1038.223,81.605,-90.860,169.523,39.682,157.462
C05263=1038.230,81.854,-90.879,169.526,39.683,157.462
C05264=1038.235,82.102,-90.897,169.528,39.683,157.462
C05265=1038.241,82.352,-90.916,169.530,39.683,157.463
C05266=1038.248,82.601,-90.935,169.532,39.684,157.463
C05267=1038.254,82.850,-90.954,169.534,39.683,157.463
C05268=1038.260,83.099,-90.972,169.536,39.684,157.463
C05269=1038.266,83.349,-90.990,169.538,39.684,157.463
C05270=1038.272,83.598,-91.009,169.540,39.684,157.463
C05271=1038.279,83.847,-91.028,169.542,39.685,157.463
C05272=1038.285,84.097,-91.047,169.545,39.685,157.464
C05273=1038.291,84.346,-91.065,169.547,39.685,157.464
C05274=1038.298,84.595,-91.084,169.549,39.686,157.464
C05275=1038.304,84.844,-91.103,169.551,39.685,157.464
C05276=1038.310,85.093,-91.122,169.553,39.686,157.464
C05277=1038.316,85.343,-91.141,169.555,39.686,157.464
C05278=1038.323,85.592,-91.159,169.557,39.686,157.464
C05279=1038.329,85.841,-91.178,169.558,39.687,157.464
C05280=1038.335,86.090,-91.197,169.560,39.687,157.464
C05281=1038.341,86.339,-91.216,169.562,39.687,157.465
C05282=1038.348,86.588,-91.234,169.565,39.687,157.465
C05283=1038.354,86.838,-91.253,169.567,39.687,157.465
C05284=1038.361,87.087,-91.272,169.569,39.688,157.465
C05285=1038.366,87.336,-91.291,169.571,39.688,157.465
C05286=1038.373,87.585,-91.310,169.573,39.688,157.465
C05287=1038.379,87.834,-91.328,169.575,39.689,157.465
C05288=1038.386,88.083,-91.347,169.577,39.688,157.465
C05289=1038.393,88.333,-91.366,169.579,39.689,157.465
C05290=1038.398,88.583,-91.385,169.581,39.689,157.466
C05291=1038.405,88.832,-91.404,169.583,39.689,157.466
C05292=1038.411,89.081,-91.422,169.586,39.690,157.466
C05293=1038.418,89.330,-91.441,169.588,39.689,157.466
C05294=1038.423,89.580,-91.460,169.590,39.690,157.466
C05295=1038.430,89.829,-91.479,169.592,39.690,157.466
C05296=1038.436,90.078,-91.498,169.594,39.690,157.466
C05297=1038.442,90.327,-91.517,169.596,39.691,157.466
C05298=1038.449,90.576,-91.536,169.598,39.691,157.467
C05299=1038.455,90.825,-91.555,169.600,39.691,157.467
C05300=1038.461,91.074,-91.574,169.602,39.691,157.467
C05301=1038.467,91.323,-91.593,169.605,39.692,157.467
C05302=1038.473,91.573,-91.612,169.607,39.692,157.467
C05303=1038.480,91.821,-91.631,169.609,39.692,157.467
C05304=1038.486,92.071,-91.651,169.611,39.693,157.467
C05305=1038.492,92.321,-91.670,169.612,39.693,157.468
C05306=1038.498,92.607,-91.691,169.615,39.694,157.468
C05307=1038.505,92.892,-91.714,169.617,39.694,157.468
C05308=1038.513,93.179,-91.735,169.619,39.694,157.468
C05309=1038.520,93.464,-91.758,169.621,39.694,157.468
C05310=1038.526,93.713,-91.776,169.624,39.695,157.468
C05311=1038.532,93.963,-91.796,169.626,39.695,157.468
C05312=1038.539,94.211,-91.815,169.628,39.695,157.468
C05313=1038.545,94.461,-91.834,169.630,39.696,157.469
C05314=1038.552,94.711,-91.853,169.632,39.696,157.469
C05315=1038.557,94.960,-91.873,169.634,39.696,157.469
C05316=1038.564,95.208,-91.892,169.636,39.696,157.469
C05317=1038.570,95.458,-91.911,169.638,39.697,157.469
C05318=1038.575,95.707,-91.930,169.640,39.697,157.469
C05319=1038.582,95.956,-91.950,169.643,39.697,157.469
C05320=1038.588,96.205,-91.969,169.645,39.698,157.470
C05321=1038.595,96.455,-91.988,169.647,39.698,157.470
C05322=1038.601,96.704,-92.008,169.649,39.698,157.470
C05323=1038.607,96.953,-92.027,169.651,39.698,157.470
C05324=1038.613,97.202,-92.046,169.653,39.699,157.470
C05325=1038.620,97.451,-92.065,169.655,39.699,157.470
C05326=1038.625,97.700,-92.084,169.657,39.699,157.470
C05327=1038.633,97.950,-92.104,169.660,39.700,157.470
C05328=1038.638,98.199,-92.123,169.662,39.700,157.471
C05329=1038.645,98.448,-92.142,169.664,39.700,157.471
C05330=1038.651,98.697,-92.162,169.666,39.701,157.471
C05331=1038.657,98.946,-92.181,169.668,39.700,157.471
C05332=1038.664,99.196,-92.201,169.670,39.701,157.471
C05333=1038.670,99.445,-92.220,169.672,39.701,157.471
C05334=1038.676,99.694,-92.239,169.674,39.701,157.471
C05335=1038.683,99.943,-92.258,169.676,39.702,157.471
C05336=1038.688,100.192,-92.278,169.679,39.702,157.472
C05337=1038.695,100.442,-92.298,169.681,39.702,157.472
C05338=1038.701,100.691,-92.317,169.683,39.702,157.472
C05339=1038.707,100.940,-92.336,169.684,39.703,157.472
C05340=1038.713,101.189,-92.356,169.686,39.703,157.472
C05341=1038.719,101.438,-92.376,169.688,39.704,157.472
C05342=1038.725,101.687,-92.396,169.690,39.704,157.472
C05343=1038.732,101.936,-92.415,169.692,39.704,157.473
C05344=1038.738,102.185,-92.435,169.694,39.705,157.473
C05345=1038.744,102.435,-92.454,169.697,39.705,157.473
C05346=1038.750,102.684,-92.474,169.699,39.706,157.473
C05347=1038.756,102.934,-92.493,169.701,39.705,157.473
C05348=1038.763,103.182,-92.513,169.703,39.706,157.473
C05349=1038.769,103.431,-92.533,169.705,39.706,157.473
C05350=1038.774,103.680,-92.552,169.707,39.707,157.474
C05351=1038.780,103.929,-92.572,169.709,39.707,157.474
C05352=1038.787,104.179,-92.592,169.711,39.707,157.474
C05353=1038.793,104.428,-92.611,169.714,39.708,157.474
C05354=1038.799,104.677,-92.631,169.716,39.708,157.474
C05355=1038.805,104.925,-92.651,169.718,39.708,157.474
C05356=1038.812,105.176,-92.670,169.720,39.709,157.474
C05357=1038.818,105.424,-92.690,169.722,39.709,157.474
C05358=1038.825,105.673,-92.710,169.724,39.709,157.475
C05359=1038.830,105.922,-92.729,169.726,39.710,157.475
C05360=1038.837,106.172,-92.749,169.729,39.710,157.475
C05361=1038.843,106.421,-92.769,169.731,39.710,157.475
C05362=1038.848,106.670,-92.789,169.733,39.710,157.475
C05363=1038.855,106.920,-92.809,169.735,39.711,157.475
C05364=1038.862,107.168,-92.828,169.737,39.711,157.476
C05365=1038.867,107.418,-92.847,169.739,39.711,157.476
C05366=1038.874,107.667,-92.868,169.741,39.712,157.476
C05367=1038.880,107.916,-92.888,169.743,39.712,157.476
C05368=1038.886,108.165,-92.908,169.745,39.713,157.476
C05369=1038.892,108.414,-92.927,169.747,39.712,157.476
C05370=1038.900,108.701,-92.950,169.750,39.713,157.476
C05371=1038.907,108.986,-92.973,169.752,39.713,157.476
C05372=1038.914,109.272,-92.996,169.755,39.714,157.477
C05373=1038.921,109.558,-93.019,169.757,39.714,157.477
C05374=1038.927,109.807,-93.037,169.759,39.715,157.477
C05375=1038.934,110.056,-93.058,169.761,39.715,157.477
C05376=1038.940,110.305,-93.078,169.763,39.715,157.477
C05377=1038.947,110.555,-93.098,169.766,39.716,157.477
C05378=1038.953,110.803,-93.118,169.768,39.716,157.478
C05379=1038.959,111.052,-93.138,169.770,39.716,157.478
C05380=1038.965,111.302,-93.158,169.772,39.716,157.478
C05381=1038.971,111.551,-93.177,169.774,39.717,157.478
C05382=1038.977,111.800,-93.197,169.776,39.717,157.478
C05383=1038.983,112.050,-93.218,169.778,39.718,157.478
C05384=1038.989,112.298,-93.238,169.781,39.718,157.478
C05385=1038.995,112.547,-93.258,169.783,39.719,157.479
C05386=1039.002,112.797,-93.278,169.785,39.718,157.479
C05387=1039.008,113.045,-93.298,169.787,39.719,157.479
C05388=1039.014,113.294,-93.318,169.789,39.719,157.479
C05389=1039.021,113.544,-93.338,169.791,39.720,157.479
C05390=1039.027,113.793,-93.358,169.793,39.720,157.479
C05391=1039.032,114.042,-93.379,169.795,39.721,157.479
C05392=1039.038,114.291,-93.399,169.798,39.721,157.480
C05393=1039.044,114.540,-93.419,169.800,39.722,157.480
C05394=1039.051,114.790,-93.439,169.802,39.722,157.480
C05395=1039.056,115.039,-93.460,169.804,39.723,157.480
C05396=1039.062,115.288,-93.480,169.806,39.723,157.480
C05397=1039.069,115.537,-93.500,169.808,39.723,157.480
C05398=1039.075,115.786,-93.520,169.810,39.723,157.481
C05399=1039.080,116.035,-93.541,169.813,39.724,157.481
C05400=1039.087,116.284,-93.562,169.815,39.724,157.481
C05401=1039.093,116.533,-93.582,169.817,39.725,157.481
C05402=1039.099,116.781,-93.602,169.818,39.725,157.481
C05403=1039.105,117.031,-93.622,169.820,39.726,157.481
C05404=1039.111,117.280,-93.642,169.822,39.726,157.482
C05405=1039.117,117.530,-93.663,169.824,39.727,157.482
C05406=1039.123,117.779,-93.683,169.827,39.727,157.482
C05407=1039.129,118.028,-93.703,169.829,39.728,157.482
C05408=1039.136,118.276,-93.724,169.831,39.728,157.482
C05409=1039.142,118.525,-93.744,169.833,39.729,157.482
C05410=1039.147,118.775,-93.765,169.835,39.729,157.483
C05411=1039.153,119.024,-93.785,169.837,39.730,157.483
C05412=1039.160,119.273,-93.805,169.840,39.730,157.483
C05413=1039.166,119.522,-93.827,169.842,39.730,157.483
C05414=1039.172,119.771,-93.847,169.844,39.730,157.483
C05415=1039.178,120.020,-93.867,169.846,39.731,157.483
C05416=1039.184,120.269,-93.887,169.848,39.731,157.483
C05417=1039.190,120.519,-93.908,169.851,39.732,157.484
C05418=1039.196,120.767,-93.929,169.853,39.732,157.484
C05419=1039.203,121.017,-93.949,169.856,39.733,157.484
C05420=1039.208,121.266,-93.969,169.858,39.733,157.484
C05421=1039.215,121.515,-93.990,169.860,39.733,157.484
C05422=1039.221,121.763,-94.010,169.862,39.734,157.484
C05423=1039.228,122.013,-94.031,169.864,39.734,157.485
C05424=1039.233,122.262,-94.051,169.866,39.735,157.485
C05425=1039.240,122.512,-94.072,169.868,39.735,157.485
C05426=1039.246,122.760,-94.092,169.870,39.735,157.485
C05427=1039.252,123.010,-94.113,169.873,39.736,157.485
